Yaskawa INFORM job: DEMO_ROOF_SIDE_0625_3PAINT_27.JBI

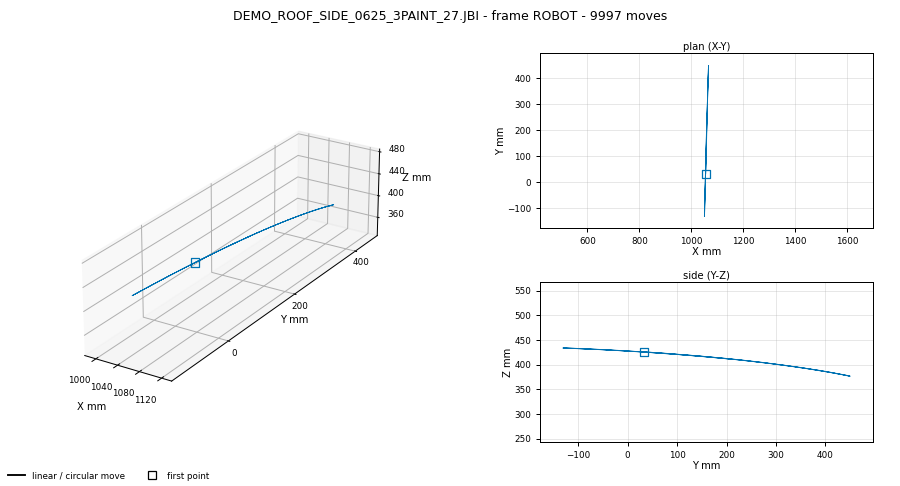
[picture p0: tool path of DEMO_ROOF_SIDE_0625_3PAINT_27.JBI in frame ROBOT, 9997 of 9997 moves have a stored position in this frame; points joined in program order, loops and branches not executed]
/JOB
//NAME DEMO_ROOF_SIDE_0625_3PAINT27
//POS
///NPOS 9997,0,0,0,0,0
///TOOL 0
///USER 0
///POSTYPE ROBOT
///RECTAN
///RCONF 1,0,0,0,0,0,0,0,0,0,0,0,0,0,0,0,0,0,0,0,0,0,0,0
C00000=1055.838,33.048,426.241,171.218,30.645,155.735
C00001=1055.844,33.297,426.225,171.220,30.647,155.735
C00002=1055.850,33.546,426.209,171.221,30.649,155.735
C00003=1055.856,33.796,426.193,171.222,30.652,155.736
C00004=1055.862,34.045,426.176,171.224,30.654,155.736
C00005=1055.869,34.295,426.160,171.225,30.656,155.736
C00006=1055.875,34.544,426.144,171.227,30.658,155.737
C00007=1055.881,34.793,426.128,171.229,30.661,155.737
C00008=1055.887,35.043,426.111,171.230,30.663,155.737
C00009=1055.893,35.292,426.095,171.231,30.665,155.738
C00010=1055.900,35.541,426.080,171.233,30.667,155.738
C00011=1055.906,35.790,426.063,171.235,30.670,155.738
C00012=1055.912,36.040,426.047,171.237,30.672,155.739
C00013=1055.918,36.290,426.030,171.237,30.674,155.739
C00014=1055.924,36.539,426.014,171.239,30.676,155.739
C00015=1055.930,36.789,425.998,171.241,30.679,155.740
C00016=1055.937,37.038,425.982,171.243,30.681,155.740
C00017=1055.943,37.287,425.966,171.244,30.683,155.740
C00018=1055.950,37.537,425.949,171.246,30.686,155.741
C00019=1055.955,37.786,425.933,171.247,30.688,155.741
C00020=1055.961,38.036,425.917,171.248,30.690,155.741
C00021=1055.967,38.285,425.901,171.250,30.693,155.742
C00022=1055.973,38.534,425.884,171.252,30.695,155.742
C00023=1055.979,38.784,425.868,171.254,30.698,155.742
C00024=1055.986,39.033,425.851,171.254,30.699,155.743
C00025=1055.992,39.282,425.835,171.256,30.702,155.743
C00026=1055.998,39.532,425.818,171.258,30.704,155.743
C00027=1056.004,39.781,425.802,171.260,30.706,155.744
C00028=1056.010,40.031,425.786,171.261,30.709,155.744
C00029=1056.016,40.280,425.769,171.263,30.711,155.744
C00030=1056.023,40.529,425.752,171.264,30.714,155.745
C00031=1056.029,40.779,425.736,171.265,30.716,155.745
C00032=1056.035,41.028,425.720,171.267,30.719,155.746
C00033=1056.041,41.277,425.703,171.269,30.721,155.746
C00034=1056.047,41.527,425.687,171.271,30.723,155.746
C00035=1056.053,41.776,425.670,171.271,30.725,155.747
C00036=1056.059,42.025,425.654,171.273,30.727,155.747
C00037=1056.065,42.275,425.637,171.275,30.730,155.747
C00038=1056.071,42.525,425.620,171.276,30.732,155.748
C00039=1056.076,42.774,425.604,171.278,30.735,155.748
C00040=1056.083,43.023,425.587,171.280,30.737,155.748
C00041=1056.089,43.273,425.571,171.281,30.739,155.749
C00042=1056.095,43.522,425.554,171.282,30.742,155.749
C00043=1056.101,43.771,425.538,171.284,30.744,155.749
C00044=1056.108,44.021,425.521,171.286,30.746,155.750
C00045=1056.113,44.270,425.504,171.287,30.748,155.750
C00046=1056.119,44.520,425.488,171.288,30.751,155.750
C00047=1056.125,44.768,425.471,171.290,30.754,155.751
C00048=1056.131,45.018,425.454,171.292,30.756,155.751
C00049=1056.137,45.268,425.437,171.293,30.759,155.752
C00050=1056.144,45.553,425.418,171.295,30.761,155.752
C00051=1056.151,45.838,425.399,171.296,30.764,155.752
C00052=1056.158,46.123,425.380,171.298,30.767,155.753
C00053=1056.164,46.410,425.360,171.300,30.769,155.753
C00054=1056.171,46.659,425.343,171.302,30.772,155.753
C00055=1056.177,46.908,425.327,171.303,30.774,155.754
C00056=1056.183,47.157,425.310,171.305,30.776,155.754
C00057=1056.189,47.407,425.293,171.306,30.779,155.755
C00058=1056.195,47.656,425.277,171.308,30.782,155.755
C00059=1056.201,47.905,425.260,171.309,30.784,155.755
C00060=1056.206,48.155,425.243,171.311,30.786,155.756
C00061=1056.213,48.404,425.226,171.313,30.788,155.756
C00062=1056.219,48.653,425.209,171.313,30.791,155.756
C00063=1056.225,48.903,425.192,171.315,30.793,155.757
C00064=1056.231,49.153,425.175,171.317,30.796,155.757
C00065=1056.237,49.401,425.158,171.319,30.798,155.757
C00066=1056.243,49.651,425.142,171.320,30.800,155.758
C00067=1056.249,49.900,425.124,171.322,30.803,155.758
C00068=1056.255,50.150,425.108,171.323,30.805,155.758
C00069=1056.262,50.398,425.091,171.324,30.807,155.759
C00070=1056.267,50.648,425.074,171.326,30.810,155.759
C00071=1056.274,50.898,425.057,171.328,30.812,155.759
C00072=1056.280,51.147,425.040,171.329,30.815,155.760
C00073=1056.285,51.396,425.023,171.330,30.817,155.760
C00074=1056.292,51.646,425.006,171.332,30.819,155.761
C00075=1056.298,51.895,424.989,171.334,30.822,155.761
C00076=1056.303,52.144,424.972,171.335,30.824,155.761
C00077=1056.310,52.394,424.955,171.337,30.827,155.762
C00078=1056.316,52.643,424.939,171.339,30.829,155.762
C00079=1056.321,52.892,424.921,171.339,30.831,155.762
C00080=1056.328,53.142,424.904,171.341,30.834,155.763
C00081=1056.334,53.391,424.887,171.343,30.836,155.763
C00082=1056.340,53.640,424.870,171.345,30.838,155.763
C00083=1056.346,53.890,424.853,171.346,30.841,155.764
C00084=1056.352,54.139,424.836,171.347,30.843,155.764
C00085=1056.359,54.389,424.818,171.349,30.846,155.765
C00086=1056.365,54.638,424.802,171.350,30.848,155.765
C00087=1056.370,54.887,424.785,171.352,30.850,155.765
C00088=1056.377,55.136,424.767,171.354,30.853,155.766
C00089=1056.383,55.386,424.751,171.356,30.855,155.766
C00090=1056.389,55.635,424.733,171.356,30.857,155.766
C00091=1056.395,55.884,424.716,171.358,30.860,155.767
C00092=1056.401,56.134,424.700,171.360,30.862,155.767
C00093=1056.407,56.383,424.682,171.361,30.865,155.767
C00094=1056.414,56.632,424.665,171.363,30.867,155.768
C00095=1056.420,56.882,424.648,171.365,30.869,155.768
C00096=1056.426,57.131,424.631,171.366,30.871,155.768
C00097=1056.433,57.381,424.613,171.367,30.873,155.769
C00098=1056.438,57.630,424.597,171.369,30.876,155.769
C00099=1056.444,57.879,424.580,171.371,30.878,155.769
C00100=1056.450,58.129,424.562,171.372,30.881,155.770
C00101=1056.457,58.377,424.545,171.374,30.883,155.770
C00102=1056.463,58.627,424.528,171.375,30.886,155.770
C00103=1056.469,58.876,424.510,171.376,30.888,155.771
C00104=1056.475,59.126,424.493,171.378,30.890,155.771
C00105=1056.481,59.375,424.476,171.380,30.892,155.771
C00106=1056.488,59.624,424.458,171.382,30.895,155.772
C00107=1056.494,59.874,424.442,171.383,30.897,155.772
C00108=1056.500,60.123,424.424,171.384,30.900,155.773
C00109=1056.506,60.372,424.407,171.386,30.902,155.773
C00110=1056.512,60.622,424.389,171.387,30.904,155.773
C00111=1056.519,60.871,424.372,171.389,30.906,155.774
C00112=1056.525,61.121,424.356,171.391,30.909,155.774
C00113=1056.531,61.370,424.338,171.392,30.911,155.774
C00114=1056.539,61.655,424.318,171.394,30.914,155.775
C00115=1056.545,61.940,424.298,171.396,30.917,155.775
C00116=1056.553,62.225,424.278,171.398,30.919,155.775
C00117=1056.559,62.510,424.259,171.399,30.922,155.776
C00118=1056.566,62.760,424.241,171.401,30.924,155.776
C00119=1056.572,63.009,424.224,171.402,30.927,155.777
C00120=1056.579,63.258,424.206,171.404,30.929,155.777
C00121=1056.584,63.507,424.189,171.405,30.931,155.777
C00122=1056.591,63.757,424.171,171.407,30.934,155.778
C00123=1056.596,64.006,424.155,171.409,30.936,155.778
C00124=1056.603,64.256,424.137,171.410,30.938,155.778
C00125=1056.609,64.505,424.120,171.411,30.941,155.779
C00126=1056.615,64.754,424.102,171.413,30.943,155.779
C00127=1056.621,65.003,424.085,171.415,30.946,155.779
C00128=1056.627,65.253,424.067,171.416,30.948,155.780
C00129=1056.634,65.502,424.050,171.418,30.950,155.780
C00130=1056.639,65.751,424.032,171.420,30.953,155.781
C00131=1056.646,66.001,424.014,171.420,30.955,155.781
C00132=1056.652,66.250,423.997,171.422,30.958,155.781
C00133=1056.658,66.500,423.979,171.424,30.960,155.782
C00134=1056.663,66.749,423.962,171.426,30.962,155.782
C00135=1056.670,66.998,423.944,171.427,30.964,155.782
C00136=1056.676,67.247,423.927,171.429,30.967,155.783
C00137=1056.682,67.497,423.909,171.430,30.970,155.783
C00138=1056.688,67.745,423.890,171.431,30.972,155.783
C00139=1056.695,67.995,423.873,171.433,30.974,155.784
C00140=1056.701,68.244,423.855,171.435,30.977,155.784
C00141=1056.706,68.493,423.838,171.436,30.979,155.785
C00142=1056.712,68.743,423.820,171.438,30.981,155.785
C00143=1056.719,68.992,423.803,171.439,30.984,155.785
C00144=1056.725,69.242,423.785,171.441,30.987,155.786
C00145=1056.730,69.491,423.767,171.442,30.989,155.786
C00146=1056.736,69.740,423.749,171.444,30.991,155.786
C00147=1056.743,69.990,423.732,171.446,30.993,155.787
C00148=1056.749,70.238,423.714,171.447,30.996,155.787
C00149=1056.755,70.488,423.696,171.448,30.999,155.788
C00150=1056.761,70.737,423.678,171.450,31.001,155.788
C00151=1056.767,70.987,423.660,171.452,31.003,155.788
C00152=1056.772,71.236,423.643,171.453,31.006,155.789
C00153=1056.779,71.485,423.624,171.455,31.008,155.789
C00154=1056.786,71.734,423.607,171.456,31.011,155.789
C00155=1056.791,71.983,423.589,171.457,31.013,155.790
C00156=1056.797,72.233,423.571,171.459,31.015,155.790
C00157=1056.803,72.482,423.554,171.461,31.018,155.790
C00158=1056.809,72.731,423.535,171.462,31.020,155.791
C00159=1056.815,72.981,423.517,171.464,31.023,155.791
C00160=1056.821,73.230,423.499,171.465,31.025,155.792
C00161=1056.827,73.480,423.482,171.467,31.027,155.792
C00162=1056.834,73.729,423.463,171.468,31.030,155.792
C00163=1056.840,73.978,423.446,171.470,31.032,155.793
C00164=1056.846,74.227,423.428,171.472,31.035,155.793
C00165=1056.851,74.476,423.410,171.473,31.037,155.793
C00166=1056.858,74.726,423.392,171.475,31.039,155.794
C00167=1056.864,74.975,423.374,171.476,31.042,155.794
C00168=1056.869,75.224,423.356,171.477,31.045,155.795
C00169=1056.876,75.474,423.338,171.479,31.047,155.795
C00170=1056.882,75.723,423.320,171.481,31.049,155.795
C00171=1056.887,75.972,423.302,171.483,31.051,155.796
C00172=1056.894,76.221,423.283,171.484,31.054,155.796
C00173=1056.900,76.471,423.266,171.485,31.057,155.796
C00174=1056.906,76.720,423.249,171.487,31.059,155.797
C00175=1056.913,76.969,423.230,171.488,31.061,155.797
C00176=1056.919,77.219,423.212,171.490,31.063,155.797
C00177=1056.925,77.468,423.193,171.492,31.066,155.798
C00178=1056.932,77.752,423.173,171.494,31.069,155.798
C00179=1056.938,78.038,423.152,171.495,31.071,155.799
C00180=1056.945,78.323,423.131,171.497,31.075,155.799
C00181=1056.952,78.608,423.111,171.499,31.077,155.800
C00182=1056.958,78.856,423.093,171.500,31.079,155.800
C00183=1056.964,79.106,423.075,171.502,31.082,155.800
C00184=1056.970,79.356,423.057,171.504,31.085,155.801
C00185=1056.976,79.605,423.037,171.505,31.087,155.801
C00186=1056.982,79.854,423.020,171.506,31.089,155.801
C00187=1056.988,80.103,423.001,171.508,31.092,155.802
C00188=1056.994,80.353,422.983,171.510,31.095,155.802
C00189=1057.000,80.602,422.965,171.511,31.097,155.803
C00190=1057.006,80.851,422.947,171.513,31.099,155.803
C00191=1057.012,81.101,422.928,171.514,31.102,155.803
C00192=1057.017,81.350,422.910,171.515,31.105,155.804
C00193=1057.024,81.599,422.892,171.517,31.107,155.804
C00194=1057.030,81.848,422.873,171.519,31.109,155.805
C00195=1057.036,82.097,422.855,171.521,31.112,155.805
C00196=1057.042,82.346,422.837,171.522,31.114,155.805
C00197=1057.047,82.596,422.818,171.523,31.117,155.806
C00198=1057.054,82.845,422.800,171.525,31.119,155.806
C00199=1057.059,83.094,422.782,171.526,31.121,155.806
C00200=1057.066,83.344,422.763,171.528,31.124,155.807
C00201=1057.072,83.593,422.745,171.530,31.127,155.807
C00202=1057.078,83.842,422.727,171.532,31.129,155.807
C00203=1057.084,84.091,422.708,171.532,31.131,155.808
C00204=1057.090,84.341,422.690,171.534,31.134,155.808
C00205=1057.096,84.590,422.671,171.536,31.136,155.809
C00206=1057.102,84.839,422.653,171.537,31.139,155.809
C00207=1057.108,85.088,422.635,171.539,31.141,155.809
C00208=1057.114,85.338,422.616,171.541,31.143,155.810
C00209=1057.120,85.587,422.597,171.543,31.146,155.810
C00210=1057.126,85.837,422.579,171.543,31.149,155.811
C00211=1057.133,86.086,422.561,171.545,31.151,155.811
C00212=1057.138,86.334,422.542,171.547,31.153,155.811
C00213=1057.144,86.584,422.524,171.548,31.156,155.812
C00214=1057.150,86.833,422.505,171.550,31.158,155.812
C00215=1057.157,87.082,422.486,171.552,31.161,155.812
C00216=1057.163,87.331,422.468,171.553,31.163,155.813
C00217=1057.169,87.582,422.449,171.554,31.165,155.813
C00218=1057.174,87.830,422.431,171.556,31.168,155.814
C00219=1057.181,88.079,422.412,171.558,31.171,155.814
C00220=1057.187,88.329,422.394,171.559,31.173,155.814
C00221=1057.193,88.578,422.376,171.561,31.175,155.815
C00222=1057.199,88.827,422.357,171.562,31.178,155.815
C00223=1057.205,89.076,422.338,171.564,31.180,155.815
C00224=1057.211,89.325,422.320,171.565,31.183,155.816
C00225=1057.217,89.575,422.302,171.567,31.185,155.816
C00226=1057.223,89.824,422.282,171.569,31.187,155.817
C00227=1057.229,90.073,422.264,171.571,31.190,155.817
C00228=1057.236,90.322,422.245,171.572,31.192,155.817
C00229=1057.242,90.571,422.227,171.573,31.195,155.818
C00230=1057.248,90.821,422.208,171.575,31.197,155.818
C00231=1057.254,91.071,422.189,171.576,31.200,155.819
C00232=1057.259,91.319,422.170,171.578,31.202,155.819
C00233=1057.266,91.568,422.152,171.580,31.205,155.819
C00234=1057.271,91.818,422.133,171.582,31.207,155.820
C00235=1057.278,92.067,422.114,171.582,31.210,155.820
C00236=1057.283,92.316,422.095,171.584,31.212,155.820
C00237=1057.290,92.566,422.076,171.586,31.214,155.821
C00238=1057.295,92.814,422.057,171.588,31.217,155.821
C00239=1057.301,93.064,422.039,171.589,31.220,155.822
C00240=1057.307,93.313,422.020,171.591,31.222,155.822
C00241=1057.313,93.563,422.001,171.593,31.224,155.822
C00242=1057.320,93.848,421.979,171.594,31.227,155.823
C00243=1057.327,94.133,421.957,171.596,31.230,155.823
C00244=1057.334,94.417,421.936,171.598,31.233,155.824
C00245=1057.340,94.702,421.915,171.600,31.236,155.824
C00246=1057.346,94.952,421.896,171.601,31.238,155.825
C00247=1057.353,95.201,421.877,171.603,31.241,155.825
C00248=1057.358,95.450,421.858,171.604,31.244,155.825
C00249=1057.365,95.699,421.839,171.606,31.246,155.826
C00250=1057.370,95.949,421.820,171.607,31.248,155.826
C00251=1057.377,96.198,421.801,171.609,31.251,155.826
C00252=1057.382,96.447,421.782,171.611,31.253,155.827
C00253=1057.389,96.696,421.764,171.612,31.255,155.827
C00254=1057.394,96.944,421.744,171.614,31.258,155.828
C00255=1057.401,97.194,421.725,171.615,31.261,155.828
C00256=1057.406,97.443,421.706,171.617,31.263,155.828
C00257=1057.413,97.692,421.687,171.618,31.265,155.829
C00258=1057.418,97.942,421.668,171.620,31.268,155.829
C00259=1057.425,98.191,421.649,171.622,31.270,155.829
C00260=1057.431,98.440,421.630,171.624,31.273,155.830
C00261=1057.437,98.689,421.612,171.624,31.275,155.830
C00262=1057.443,98.939,421.592,171.626,31.278,155.831
C00263=1057.449,99.188,421.574,171.628,31.280,155.831
C00264=1057.455,99.437,421.554,171.630,31.283,155.831
C00265=1057.461,99.686,421.535,171.631,31.285,155.832
C00266=1057.467,99.935,421.516,171.633,31.287,155.832
C00267=1057.473,100.185,421.497,171.635,31.290,155.833
C00268=1057.479,100.434,421.478,171.636,31.293,155.833
C00269=1057.485,100.683,421.459,171.637,31.295,155.833
C00270=1057.491,100.932,421.440,171.639,31.297,155.834
C00271=1057.497,101.181,421.420,171.641,31.300,155.834
C00272=1057.503,101.431,421.401,171.643,31.303,155.835
C00273=1057.509,101.680,421.382,171.644,31.305,155.835
C00274=1057.515,101.929,421.363,171.646,31.307,155.835
C00275=1057.521,102.178,421.343,171.647,31.310,155.836
C00276=1057.527,102.427,421.324,171.649,31.313,155.836
C00277=1057.533,102.677,421.305,171.650,31.315,155.837
C00278=1057.539,102.926,421.286,171.652,31.318,155.837
C00279=1057.545,103.175,421.266,171.654,31.320,155.837
C00280=1057.551,103.424,421.247,171.656,31.322,155.838
C00281=1057.556,103.674,421.227,171.657,31.325,155.838
C00282=1057.562,103.923,421.208,171.658,31.328,155.839
C00283=1057.569,104.172,421.189,171.660,31.330,155.839
C00284=1057.575,104.421,421.170,171.662,31.332,155.839
C00285=1057.580,104.670,421.150,171.663,31.335,155.840
C00286=1057.586,104.919,421.130,171.665,31.338,155.840
C00287=1057.592,105.169,421.111,171.667,31.340,155.840
C00288=1057.598,105.418,421.092,171.669,31.343,155.841
C00289=1057.604,105.667,421.073,171.669,31.345,155.841
C00290=1057.610,105.916,421.053,171.671,31.348,155.842
C00291=1057.616,106.165,421.033,171.673,31.350,155.842
C00292=1057.622,106.414,421.014,171.675,31.353,155.842
C00293=1057.628,106.663,420.995,171.676,31.355,155.843
C00294=1057.634,106.912,420.975,171.678,31.357,155.843
C00295=1057.640,107.162,420.956,171.680,31.360,155.844
C00296=1057.646,107.410,420.936,171.681,31.363,155.844
C00297=1057.651,107.660,420.917,171.682,31.365,155.844
C00298=1057.659,107.910,420.898,171.684,31.367,155.845
C00299=1057.665,108.158,420.878,171.686,31.370,155.845
C00300=1057.670,108.408,420.859,171.688,31.373,155.846
C00301=1057.676,108.657,420.839,171.689,31.375,155.846
C00302=1057.682,108.906,420.820,171.691,31.377,155.846
C00303=1057.688,109.155,420.800,171.692,31.380,155.847
C00304=1057.694,109.404,420.781,171.694,31.383,155.847
C00305=1057.700,109.653,420.761,171.695,31.385,155.848
C00306=1057.707,109.938,420.739,171.698,31.388,155.848
C00307=1057.714,110.224,420.716,171.700,31.391,155.848
C00308=1057.721,110.508,420.693,171.702,31.393,155.849
C00309=1057.728,110.793,420.671,171.703,31.396,155.849
C00310=1057.734,111.042,420.652,171.704,31.398,155.850
C00311=1057.740,111.292,420.632,171.706,31.401,155.850
C00312=1057.745,111.540,420.612,171.708,31.404,155.850
C00313=1057.751,111.790,420.593,171.710,31.406,155.851
C00314=1057.757,112.039,420.573,171.711,31.409,155.851
C00315=1057.763,112.289,420.553,171.713,31.411,155.852
C00316=1057.769,112.538,420.534,171.714,31.414,155.852
C00317=1057.775,112.786,420.514,171.716,31.416,155.852
C00318=1057.781,113.036,420.494,171.718,31.419,155.853
C00319=1057.787,113.285,420.474,171.719,31.421,155.853
C00320=1057.793,113.534,420.455,171.721,31.423,155.854
C00321=1057.799,113.783,420.435,171.723,31.426,155.854
C00322=1057.805,114.032,420.415,171.725,31.429,155.854
C00323=1057.811,114.282,420.396,171.726,31.431,155.855
C00324=1057.817,114.531,420.376,171.727,31.434,155.855
C00325=1057.823,114.779,420.356,171.729,31.437,155.856
C00326=1057.829,115.029,420.336,171.731,31.439,155.856
C00327=1057.834,115.278,420.316,171.733,31.442,155.857
C00328=1057.840,115.527,420.296,171.734,31.444,155.857
C00329=1057.846,115.776,420.276,171.736,31.446,155.857
C00330=1057.852,116.026,420.256,171.738,31.449,155.858
C00331=1057.858,116.275,420.236,171.739,31.452,155.858
C00332=1057.864,116.524,420.216,171.740,31.454,155.859
C00333=1057.870,116.772,420.196,171.742,31.457,155.859
C00334=1057.875,117.022,420.177,171.744,31.460,155.859
C00335=1057.881,117.271,420.157,171.746,31.462,155.860
C00336=1057.887,117.521,420.136,171.748,31.465,155.860
C00337=1057.893,117.769,420.116,171.749,31.467,155.861
C00338=1057.899,118.018,420.096,171.750,31.470,155.861
C00339=1057.905,118.268,420.077,171.752,31.472,155.861
C00340=1057.910,118.517,420.056,171.754,31.475,155.862
C00341=1057.916,118.766,420.036,171.756,31.477,155.862
C00342=1057.923,119.015,420.016,171.757,31.480,155.863
C00343=1057.929,119.264,419.996,171.759,31.483,155.863
C00344=1057.934,119.513,419.975,171.761,31.485,155.863
C00345=1057.940,119.762,419.956,171.762,31.488,155.864
C00346=1057.946,120.011,419.936,171.764,31.491,155.864
C00347=1057.952,120.261,419.916,171.765,31.493,155.865
C00348=1057.957,120.510,419.895,171.767,31.495,155.865
C00349=1057.963,120.759,419.875,171.769,31.498,155.865
C00350=1057.969,121.008,419.855,171.771,31.500,155.866
C00351=1057.976,121.257,419.835,171.773,31.503,155.866
C00352=1057.981,121.506,419.814,171.774,31.506,155.867
C00353=1057.987,121.755,419.794,171.775,31.508,155.867
C00354=1057.993,122.004,419.774,171.777,31.511,155.868
C00355=1057.999,122.254,419.754,171.779,31.513,155.868
C00356=1058.005,122.502,419.734,171.781,31.516,155.868
C00357=1058.011,122.751,419.714,171.782,31.518,155.869
C00358=1058.017,123.000,419.694,171.784,31.521,155.869
C00359=1058.023,123.250,419.673,171.786,31.523,155.870
C00360=1058.029,123.499,419.654,171.787,31.526,155.870
C00361=1058.035,123.748,419.634,171.789,31.529,155.870
C00362=1058.040,123.998,419.613,171.790,31.531,155.871
C00363=1058.047,124.246,419.592,171.792,31.533,155.871
C00364=1058.053,124.495,419.572,171.794,31.536,155.872
C00365=1058.059,124.744,419.552,171.796,31.539,155.872
C00366=1058.065,124.994,419.531,171.798,31.541,155.872
C00367=1058.071,125.242,419.511,171.800,31.544,155.873
C00368=1058.077,125.491,419.491,171.800,31.546,155.873
C00369=1058.082,125.741,419.470,171.802,31.548,155.874
C00370=1058.090,126.025,419.448,171.804,31.552,155.874
C00371=1058.096,126.310,419.424,171.806,31.554,155.874
C00372=1058.103,126.595,419.401,171.809,31.558,155.875
C00373=1058.110,126.880,419.378,171.811,31.560,155.875
C00374=1058.116,127.130,419.357,171.812,31.563,155.876
C00375=1058.122,127.378,419.337,171.813,31.565,155.876
C00376=1058.128,127.627,419.317,171.815,31.567,155.877
C00377=1058.134,127.877,419.296,171.817,31.570,155.877
C00378=1058.140,128.126,419.276,171.819,31.573,155.877
C00379=1058.146,128.374,419.256,171.821,31.575,155.878
C00380=1058.152,128.624,419.235,171.823,31.578,155.878
C00381=1058.158,128.873,419.215,171.824,31.580,155.879
C00382=1058.165,129.122,419.194,171.826,31.583,155.879
C00383=1058.170,129.371,419.174,171.827,31.585,155.879
C00384=1058.176,129.620,419.153,171.829,31.588,155.880
C00385=1058.182,129.869,419.132,171.831,31.591,155.880
C00386=1058.188,130.118,419.112,171.833,31.593,155.881
C00387=1058.195,130.368,419.092,171.834,31.595,155.881
C00388=1058.200,130.617,419.071,171.836,31.598,155.881
C00389=1058.207,130.866,419.050,171.838,31.600,155.882
C00390=1058.213,131.115,419.030,171.840,31.603,155.882
C00391=1058.218,131.364,419.010,171.841,31.606,155.883
C00392=1058.225,131.613,418.989,171.843,31.608,155.883
C00393=1058.230,131.862,418.968,171.845,31.610,155.883
C00394=1058.237,132.111,418.948,171.846,31.613,155.884
C00395=1058.242,132.360,418.927,171.848,31.615,155.884
C00396=1058.248,132.609,418.907,171.850,31.618,155.885
C00397=1058.254,132.858,418.886,171.852,31.621,155.885
C00398=1058.259,133.107,418.865,171.854,31.623,155.885
C00399=1058.266,133.356,418.844,171.855,31.626,155.886
C00400=1058.272,133.606,418.824,171.857,31.629,155.886
C00401=1058.277,133.855,418.803,171.858,31.631,155.887
C00402=1058.284,134.104,418.782,171.860,31.634,155.887
C00403=1058.289,134.353,418.761,171.862,31.636,155.888
C00404=1058.296,134.602,418.740,171.864,31.639,155.888
C00405=1058.301,134.851,418.720,171.866,31.642,155.888
C00406=1058.307,135.100,418.698,171.868,31.644,155.889
C00407=1058.313,135.349,418.678,171.869,31.646,155.889
C00408=1058.319,135.599,418.657,171.871,31.649,155.890
C00409=1058.325,135.847,418.636,171.872,31.652,155.890
C00410=1058.331,136.096,418.616,171.874,31.654,155.890
C00411=1058.337,136.345,418.594,171.876,31.657,155.891
C00412=1058.342,136.594,418.574,171.878,31.659,155.891
C00413=1058.349,136.843,418.553,171.880,31.662,155.892
C00414=1058.354,137.092,418.532,171.882,31.665,155.892
C00415=1058.360,137.341,418.511,171.883,31.667,155.893
C00416=1058.366,137.590,418.491,171.885,31.670,155.893
C00417=1058.373,137.839,418.469,171.886,31.672,155.893
C00418=1058.378,138.089,418.449,171.888,31.675,155.894
C00419=1058.385,138.337,418.428,171.890,31.678,155.894
C00420=1058.390,138.587,418.407,171.892,31.680,155.895
C00421=1058.396,138.836,418.385,171.894,31.682,155.895
C00422=1058.401,139.085,418.365,171.896,31.685,155.895
C00423=1058.408,139.334,418.344,171.897,31.688,155.896
C00424=1058.414,139.582,418.322,171.899,31.690,155.896
C00425=1058.420,139.832,418.302,171.901,31.693,155.897
C00426=1058.425,140.081,418.280,171.902,31.695,155.897
C00427=1058.432,140.330,418.260,171.904,31.698,155.897
C00428=1058.437,140.579,418.239,171.906,31.701,155.898
C00429=1058.444,140.828,418.217,171.908,31.703,155.898
C00430=1058.449,141.077,418.196,171.910,31.706,155.899
C00431=1058.455,141.326,418.175,171.911,31.709,155.899
C00432=1058.461,141.575,418.154,171.913,31.711,155.900
C00433=1058.466,141.824,418.133,171.915,31.714,155.900
C00434=1058.474,142.109,418.108,171.917,31.717,155.901
C00435=1058.481,142.393,418.084,171.919,31.720,155.901
C00436=1058.487,142.678,418.059,171.921,31.723,155.901
C00437=1058.493,142.963,418.036,171.923,31.726,155.902
C00438=1058.500,143.212,418.014,171.925,31.728,155.902
C00439=1058.505,143.461,417.993,171.926,31.731,155.903
C00440=1058.511,143.710,417.971,171.928,31.733,155.903
C00441=1058.517,143.959,417.951,171.930,31.736,155.904
C00442=1058.523,144.208,417.929,171.932,31.739,155.904
C00443=1058.530,144.457,417.908,171.934,31.741,155.904
C00444=1058.535,144.706,417.887,171.936,31.744,155.905
C00445=1058.541,144.956,417.866,171.938,31.747,155.905
C00446=1058.547,145.204,417.845,171.940,31.749,155.906
C00447=1058.553,145.453,417.823,171.942,31.752,155.906
C00448=1058.559,145.702,417.802,171.942,31.754,155.907
C00449=1058.565,145.951,417.780,171.944,31.757,155.907
C00450=1058.571,146.200,417.759,171.946,31.760,155.907
C00451=1058.576,146.449,417.738,171.948,31.762,155.908
C00452=1058.582,146.698,417.716,171.950,31.765,155.908
C00453=1058.588,146.948,417.695,171.952,31.767,155.909
C00454=1058.594,147.196,417.674,171.954,31.770,155.909
C00455=1058.600,147.445,417.652,171.956,31.773,155.910
C00456=1058.607,147.694,417.631,171.957,31.775,155.910
C00457=1058.612,147.943,417.609,171.959,31.778,155.910
C00458=1058.618,148.192,417.587,171.961,31.781,155.911
C00459=1058.623,148.441,417.567,171.963,31.783,155.911
C00460=1058.629,148.691,417.545,171.965,31.786,155.912
C00461=1058.636,148.940,417.524,171.967,31.788,155.912
C00462=1058.641,149.188,417.502,171.969,31.791,155.912
C00463=1058.647,149.438,417.481,171.971,31.794,155.913
C00464=1058.653,149.687,417.459,171.972,31.797,155.913
C00465=1058.659,149.935,417.438,171.973,31.799,155.914
C00466=1058.665,150.184,417.416,171.975,31.802,155.914
C00467=1058.671,150.434,417.394,171.977,31.805,155.915
C00468=1058.676,150.683,417.373,171.979,31.807,155.915
C00469=1058.682,150.932,417.351,171.981,31.810,155.916
C00470=1058.688,151.181,417.329,171.983,31.813,155.916
C00471=1058.694,151.429,417.308,171.985,31.815,155.916
C00472=1058.700,151.679,417.286,171.987,31.818,155.917
C00473=1058.707,151.927,417.264,171.989,31.820,155.917
C00474=1058.711,152.176,417.242,171.990,31.823,155.918
C00475=1058.718,152.425,417.221,171.992,31.826,155.918
C00476=1058.724,152.674,417.199,171.994,31.828,155.919
C00477=1058.729,152.923,417.178,171.996,31.831,155.919
C00478=1058.736,153.172,417.156,171.998,31.834,155.919
C00479=1058.742,153.421,417.134,172.000,31.837,155.920
C00480=1058.747,153.671,417.112,172.002,31.839,155.920
C00481=1058.753,153.919,417.091,172.004,31.842,155.921
C00482=1058.759,154.168,417.069,172.005,31.845,155.921
C00483=1058.765,154.417,417.047,172.007,31.847,155.922
C00484=1058.771,154.666,417.026,172.009,31.850,155.922
C00485=1058.776,154.915,417.003,172.011,31.852,155.922
C00486=1058.782,155.164,416.982,172.013,31.855,155.923
C00487=1058.789,155.414,416.960,172.015,31.858,155.923
C00488=1058.794,155.661,416.938,172.017,31.860,155.924
C00489=1058.800,155.911,416.916,172.019,31.863,155.924
C00490=1058.806,156.160,416.894,172.021,31.866,155.925
C00491=1058.812,156.409,416.873,172.022,31.869,155.925
C00492=1058.817,156.658,416.850,172.024,31.871,155.926
C00493=1058.824,156.907,416.828,172.026,31.874,155.926
C00494=1058.830,157.156,416.807,172.028,31.877,155.926
C00495=1058.835,157.406,416.785,172.029,31.879,155.927
C00496=1058.841,157.653,416.763,172.031,31.882,155.927
C00497=1058.847,157.903,416.741,172.033,31.884,155.928
C00498=1058.854,158.187,416.715,172.036,31.888,155.928
C00499=1058.861,158.472,416.690,172.038,31.891,155.929
C00500=1058.867,158.756,416.665,172.039,31.894,155.929
C00501=1058.874,159.041,416.641,172.042,31.897,155.930
C00502=1058.880,159.290,416.618,172.044,31.899,155.930
C00503=1058.885,159.538,416.596,172.046,31.902,155.931
C00504=1058.892,159.787,416.574,172.048,31.905,155.931
C00505=1058.897,160.036,416.552,172.050,31.908,155.931
C00506=1058.904,160.285,416.530,172.052,31.910,155.932
C00507=1058.910,160.534,416.508,172.054,31.913,155.932
C00508=1058.915,160.783,416.486,172.056,31.916,155.933
C00509=1058.921,161.031,416.464,172.058,31.918,155.933
C00510=1058.927,161.281,416.441,172.059,31.921,155.934
C00511=1058.932,161.530,416.418,172.061,31.924,155.934
C00512=1058.939,161.779,416.397,172.063,31.927,155.935
C00513=1058.944,162.027,416.374,172.065,31.929,155.935
C00514=1058.949,162.277,416.352,172.067,31.932,155.936
C00515=1058.956,162.525,416.330,172.069,31.935,155.936
C00516=1058.961,162.775,416.307,172.071,31.938,155.936
C00517=1058.967,163.024,416.284,172.073,31.941,155.937
C00518=1058.972,163.272,416.263,172.075,31.943,155.937
C00519=1058.978,163.521,416.240,172.076,31.946,155.938
C00520=1058.984,163.771,416.218,172.078,31.949,155.938
C00521=1058.989,164.019,416.195,172.080,31.952,155.939
C00522=1058.995,164.269,416.173,172.082,31.954,155.939
C00523=1059.001,164.517,416.151,172.084,31.958,155.940
C00524=1059.006,164.766,416.128,172.086,31.960,155.940
C00525=1059.012,165.015,416.106,172.088,31.963,155.941
C00526=1059.018,165.264,416.083,172.090,31.966,155.941
C00527=1059.024,165.513,416.060,172.092,31.969,155.942
C00528=1059.029,165.762,416.039,172.093,31.971,155.942
C00529=1059.035,166.010,416.016,172.095,31.974,155.942
C00530=1059.041,166.259,415.993,172.097,31.977,155.943
C00531=1059.046,166.509,415.971,172.099,31.980,155.943
C00532=1059.052,166.758,415.948,172.101,31.982,155.944
C00533=1059.059,167.006,415.926,172.103,31.985,155.944
C00534=1059.064,167.256,415.903,172.105,31.988,155.945
C00535=1059.070,167.505,415.881,172.107,31.991,155.945
C00536=1059.075,167.753,415.858,172.109,31.994,155.946
C00537=1059.081,168.002,415.836,172.111,31.996,155.946
C00538=1059.087,168.251,415.813,172.113,31.999,155.947
C00539=1059.092,168.500,415.790,172.115,32.002,155.947
C00540=1059.098,168.749,415.767,172.117,32.005,155.948
C00541=1059.105,168.997,415.745,172.119,32.008,155.948
C00542=1059.110,169.247,415.723,172.121,32.010,155.948
C00543=1059.116,169.496,415.700,172.123,32.013,155.949
C00544=1059.122,169.744,415.677,172.125,32.016,155.949
C00545=1059.128,169.993,415.655,172.127,32.019,155.950
C00546=1059.134,170.242,415.632,172.129,32.022,155.950
C00547=1059.139,170.491,415.609,172.131,32.024,155.951
C00548=1059.145,170.740,415.587,172.132,32.027,155.951
C00549=1059.151,170.989,415.564,172.134,32.030,155.952
C00550=1059.156,171.237,415.542,172.136,32.033,155.952
C00551=1059.162,171.486,415.519,172.139,32.035,155.953
C00552=1059.168,171.735,415.496,172.141,32.038,155.953
C00553=1059.174,171.984,415.473,172.143,32.041,155.954
C00554=1059.179,172.233,415.451,172.145,32.044,155.954
C00555=1059.186,172.482,415.428,172.147,32.046,155.954
C00556=1059.191,172.731,415.405,172.149,32.050,155.955
C00557=1059.197,172.980,415.382,172.151,32.052,155.955
C00558=1059.203,173.229,415.359,172.152,32.055,155.956
C00559=1059.209,173.478,415.336,172.154,32.058,155.956
C00560=1059.215,173.726,415.314,172.156,32.061,155.957
C00561=1059.221,173.976,415.291,172.159,32.063,155.957
C00562=1059.228,174.259,415.265,172.161,32.067,155.958
C00563=1059.234,174.544,415.238,172.163,32.070,155.958
C00564=1059.241,174.828,415.213,172.166,32.073,155.959
C00565=1059.248,175.111,415.187,172.168,32.076,155.959
C00566=1059.254,175.361,415.163,172.170,32.079,155.960
C00567=1059.260,175.610,415.140,172.172,32.081,155.960
C00568=1059.265,175.859,415.118,172.174,32.085,155.961
C00569=1059.272,176.107,415.095,172.176,32.087,155.961
C00570=1059.278,176.356,415.072,172.178,32.090,155.962
C00571=1059.283,176.605,415.049,172.180,32.093,155.962
C00572=1059.289,176.854,415.026,172.182,32.096,155.963
C00573=1059.295,177.103,415.003,172.184,32.098,155.963
C00574=1059.301,177.351,414.980,172.186,32.101,155.963
C00575=1059.306,177.600,414.957,172.189,32.104,155.964
C00576=1059.314,177.849,414.934,172.191,32.107,155.964
C00577=1059.319,178.098,414.911,172.193,32.109,155.965
C00578=1059.325,178.347,414.888,172.195,32.113,155.965
C00579=1059.331,178.596,414.865,172.196,32.115,155.966
C00580=1059.336,178.845,414.842,172.198,32.118,155.966
C00581=1059.343,179.093,414.819,172.200,32.121,155.967
C00582=1059.348,179.342,414.796,172.203,32.124,155.967
C00583=1059.355,179.591,414.773,172.205,32.126,155.968
C00584=1059.361,179.840,414.750,172.207,32.129,155.968
C00585=1059.367,180.089,414.727,172.209,32.132,155.969
C00586=1059.373,180.337,414.703,172.211,32.135,155.969
C00587=1059.379,180.586,414.680,172.213,32.138,155.969
C00588=1059.385,180.836,414.657,172.216,32.140,155.970
C00589=1059.391,181.085,414.634,172.218,32.143,155.970
C00590=1059.396,181.334,414.611,172.219,32.146,155.971
C00591=1059.402,181.582,414.588,172.221,32.149,155.971
C00592=1059.408,181.831,414.565,172.223,32.151,155.972
C00593=1059.415,182.080,414.542,172.226,32.154,155.972
C00594=1059.421,182.328,414.518,172.228,32.157,155.973
C00595=1059.427,182.577,414.495,172.230,32.160,155.973
C00596=1059.433,182.826,414.472,172.232,32.162,155.974
C00597=1059.439,183.075,414.448,172.234,32.166,155.974
C00598=1059.445,183.324,414.425,172.237,32.168,155.975
C00599=1059.451,183.573,414.402,172.239,32.171,155.975
C00600=1059.457,183.821,414.379,172.241,32.174,155.975
C00601=1059.463,184.071,414.355,172.242,32.177,155.976
C00602=1059.469,184.320,414.333,172.244,32.179,155.976
C00603=1059.475,184.568,414.309,172.247,32.183,155.977
C00604=1059.481,184.817,414.286,172.249,32.185,155.977
C00605=1059.487,185.066,414.261,172.251,32.188,155.978
C00606=1059.492,185.315,414.238,172.253,32.191,155.978
C00607=1059.498,185.563,414.215,172.255,32.194,155.979
C00608=1059.503,185.813,414.191,172.257,32.197,155.979
C00609=1059.509,186.061,414.167,172.260,32.200,155.980
C00610=1059.514,186.310,414.144,172.262,32.203,155.980
C00611=1059.521,186.559,414.120,172.264,32.206,155.981
C00612=1059.527,186.808,414.097,172.265,32.209,155.981
C00613=1059.532,187.056,414.073,172.267,32.212,155.982
C00614=1059.538,187.305,414.050,172.270,32.215,155.982
C00615=1059.543,187.554,414.026,172.272,32.218,155.983
C00616=1059.550,187.803,414.001,172.274,32.221,155.983
C00617=1059.555,188.052,413.979,172.276,32.224,155.984
C00618=1059.561,188.300,413.954,172.278,32.227,155.984
C00619=1059.566,188.549,413.931,172.281,32.230,155.985
C00620=1059.572,188.798,413.907,172.283,32.233,155.985
C00621=1059.578,189.047,413.883,172.285,32.236,155.986
C00622=1059.583,189.296,413.860,172.287,32.239,155.986
C00623=1059.589,189.544,413.836,172.290,32.242,155.987
C00624=1059.595,189.793,413.812,172.291,32.245,155.987
C00625=1059.601,190.043,413.788,172.293,32.247,155.988
C00626=1059.608,190.326,413.761,172.296,32.251,155.988
C00627=1059.614,190.609,413.735,172.298,32.254,155.989
C00628=1059.621,190.893,413.707,172.301,32.258,155.990
C00629=1059.628,191.177,413.680,172.303,32.262,155.990
C00630=1059.633,191.425,413.656,172.305,32.264,155.991
C00631=1059.639,191.674,413.632,172.308,32.267,155.991
C00632=1059.646,191.923,413.608,172.310,32.271,155.992
C00633=1059.651,192.171,413.584,172.312,32.273,155.992
C00634=1059.657,192.420,413.561,172.314,32.276,155.993
C00635=1059.662,192.669,413.536,172.317,32.279,155.993
C00636=1059.669,192.918,413.512,172.318,32.282,155.994
C00637=1059.674,193.166,413.488,172.320,32.285,155.994
C00638=1059.680,193.415,413.464,172.322,32.288,155.995
C00639=1059.685,193.664,413.441,172.325,32.291,155.995
C00640=1059.692,193.913,413.417,172.327,32.294,155.996
C00641=1059.697,194.162,413.392,172.329,32.297,155.996
C00642=1059.703,194.410,413.369,172.332,32.300,155.997
C00643=1059.709,194.660,413.344,172.334,32.303,155.997
C00644=1059.715,194.908,413.320,172.336,32.306,155.998
C00645=1059.721,195.156,413.296,172.338,32.309,155.998
C00646=1059.727,195.405,413.272,172.341,32.312,155.999
C00647=1059.732,195.655,413.249,172.343,32.315,155.999
C00648=1059.739,195.904,413.225,172.344,32.318,156.000
C00649=1059.744,196.152,413.200,172.347,32.321,156.000
C00650=1059.751,196.401,413.176,172.349,32.324,156.001
C00651=1059.756,196.650,413.152,172.351,32.327,156.001
C00652=1059.762,196.898,413.128,172.353,32.330,156.002
C00653=1059.768,197.147,413.104,172.356,32.333,156.002
C00654=1059.774,197.396,413.080,172.358,32.336,156.003
C00655=1059.780,197.645,413.055,172.360,32.339,156.003
C00656=1059.786,197.893,413.032,172.363,32.342,156.004
C00657=1059.792,198.143,413.007,172.365,32.345,156.004
C00658=1059.798,198.391,412.983,172.367,32.348,156.005
C00659=1059.804,198.640,412.959,172.370,32.351,156.005
C00660=1059.810,198.888,412.935,172.372,32.354,156.006
C00661=1059.816,199.137,412.910,172.374,32.357,156.006
C00662=1059.822,199.385,412.886,172.376,32.360,156.007
C00663=1059.828,199.635,412.862,172.378,32.363,156.007
C00664=1059.833,199.883,412.837,172.380,32.366,156.008
C00665=1059.840,200.132,412.813,172.383,32.369,156.008
C00666=1059.845,200.381,412.789,172.385,32.372,156.009
C00667=1059.852,200.630,412.765,172.387,32.375,156.009
C00668=1059.857,200.878,412.741,172.390,32.378,156.010
C00669=1059.864,201.127,412.716,172.392,32.381,156.010
C00670=1059.870,201.376,412.691,172.394,32.384,156.011
C00671=1059.876,201.624,412.668,172.397,32.387,156.011
C00672=1059.882,201.874,412.643,172.399,32.391,156.012
C00673=1059.887,202.122,412.619,172.401,32.393,156.012
C00674=1059.894,202.371,412.594,172.404,32.396,156.013
C00675=1059.900,202.619,412.570,172.405,32.400,156.014
C00676=1059.905,202.868,412.545,172.407,32.403,156.014
C00677=1059.911,203.117,412.521,172.410,32.406,156.015
C00678=1059.917,203.366,412.496,172.412,32.409,156.015
C00679=1059.922,203.614,412.471,172.415,32.412,156.016
C00680=1059.928,203.863,412.447,172.417,32.415,156.016
C00681=1059.934,204.111,412.422,172.419,32.419,156.017
C00682=1059.940,204.360,412.398,172.422,32.421,156.017
C00683=1059.946,204.610,412.373,172.424,32.424,156.018
C00684=1059.952,204.858,412.348,172.426,32.428,156.018
C00685=1059.958,205.107,412.324,172.429,32.431,156.019
C00686=1059.963,205.355,412.299,172.431,32.434,156.019
C00687=1059.969,205.604,412.274,172.433,32.437,156.020
C00688=1059.975,205.853,412.250,172.436,32.440,156.021
C00689=1059.982,206.101,412.225,172.438,32.444,156.021
C00690=1060.006,207.150,412.121,172.620,32.529,156.031
C00691=1060.012,207.381,412.097,172.622,32.533,156.031
C00692=1060.017,207.611,412.073,172.623,32.536,156.032
C00693=1060.023,207.842,412.050,172.625,32.540,156.033
C00694=1060.029,208.072,412.026,172.627,32.543,156.033
C00695=1060.035,208.302,412.002,172.629,32.547,156.034
C00696=1060.040,208.532,411.978,172.631,32.551,156.035
C00697=1060.046,208.763,411.954,172.633,32.555,156.036
C00698=1060.052,208.993,411.931,172.633,32.559,156.036
C00699=1060.057,209.242,411.905,172.635,32.562,156.037
C00700=1060.064,209.490,411.879,172.637,32.567,156.038
C00701=1060.070,209.740,411.854,172.639,32.570,156.038
C00702=1060.077,209.988,411.828,172.641,32.575,156.039
C00703=1060.082,210.237,411.802,172.643,32.578,156.040
C00704=1060.089,210.485,411.776,172.645,32.583,156.041
C00705=1060.095,210.734,411.751,172.647,32.586,156.041
C00706=1060.101,210.982,411.725,172.649,32.591,156.042
C00707=1060.107,211.231,411.699,172.651,32.594,156.043
C00708=1060.113,211.480,411.674,172.653,32.599,156.044
C00709=1060.120,211.728,411.648,172.656,32.602,156.044
C00710=1060.125,211.977,411.622,172.658,32.607,156.045
C00711=1060.131,212.225,411.596,172.660,32.610,156.046
C00712=1060.138,212.473,411.570,172.662,32.615,156.047
C00713=1060.143,212.722,411.544,172.664,32.618,156.047
C00714=1060.150,212.971,411.518,172.666,32.623,156.048
C00715=1060.156,213.220,411.492,172.668,32.626,156.049
C00716=1060.162,213.468,411.466,172.670,32.630,156.049
C00717=1060.168,213.717,411.440,172.672,32.634,156.050
C00718=1060.174,213.965,411.414,172.674,32.638,156.051
C00719=1060.180,214.214,411.388,172.676,32.642,156.052
C00720=1060.186,214.462,411.362,172.677,32.646,156.052
C00721=1060.192,214.711,411.336,172.679,32.650,156.053
C00722=1060.198,214.959,411.310,172.681,32.654,156.054
C00723=1060.204,215.208,411.285,172.683,32.658,156.055
C00724=1060.211,215.457,411.258,172.685,32.662,156.055
C00725=1060.217,215.706,411.232,172.687,32.666,156.056
C00726=1060.223,215.954,411.206,172.689,32.670,156.057
C00727=1060.229,216.202,411.180,172.691,32.674,156.058
C00728=1060.235,216.451,411.154,172.693,32.678,156.058
C00729=1060.241,216.699,411.128,172.695,32.682,156.059
C00730=1060.247,216.949,411.101,172.697,32.686,156.060
C00731=1060.254,217.197,411.075,172.699,32.690,156.061
C00732=1060.260,217.445,411.049,172.701,32.694,156.061
C00733=1060.265,217.694,411.023,172.703,32.698,156.062
C00734=1060.272,217.942,410.997,172.706,32.702,156.063
C00735=1060.278,218.191,410.970,172.708,32.706,156.063
C00736=1060.284,218.440,410.944,172.710,32.709,156.064
C00737=1060.290,218.688,410.918,172.712,32.714,156.065
C00738=1060.296,218.936,410.891,172.714,32.717,156.066
C00739=1060.302,219.185,410.866,172.716,32.721,156.066
C00740=1060.309,219.434,410.839,172.718,32.725,156.067
C00741=1060.315,219.682,410.812,172.720,32.729,156.068
C00742=1060.321,219.930,410.786,172.722,32.733,156.069
C00743=1060.327,220.179,410.761,172.724,32.737,156.069
C00744=1060.334,220.428,410.734,172.726,32.741,156.070
C00745=1060.340,220.676,410.707,172.729,32.745,156.071
C00746=1060.346,220.925,410.681,172.731,32.749,156.071
C00747=1060.352,221.158,410.657,172.733,32.752,156.072
C00748=1060.357,221.391,410.632,172.735,32.756,156.073
C00749=1060.363,221.624,410.607,172.737,32.760,156.074
C00750=1060.368,221.857,410.582,172.738,32.763,156.074
C00751=1060.374,222.089,410.557,172.740,32.767,156.075
C00752=1060.380,222.322,410.532,172.742,32.771,156.076
C00753=1060.386,222.555,410.507,172.743,32.774,156.076
C00754=1060.391,222.788,410.483,172.745,32.778,156.077
C00755=1060.397,223.036,410.456,172.747,32.782,156.078
C00756=1060.404,223.285,410.429,172.750,32.786,156.078
C00757=1060.410,223.533,410.403,172.752,32.790,156.079
C00758=1060.416,223.781,410.376,172.754,32.794,156.080
C00759=1060.422,224.030,410.350,172.756,32.798,156.081
C00760=1060.428,224.279,410.323,172.758,32.802,156.081
C00761=1060.434,224.527,410.296,172.760,32.805,156.082
C00762=1060.440,224.775,410.270,172.762,32.810,156.083
C00763=1060.447,225.024,410.243,172.764,32.813,156.084
C00764=1060.452,225.273,410.216,172.767,32.818,156.084
C00765=1060.458,225.521,410.190,172.769,32.821,156.085
C00766=1060.465,225.770,410.163,172.771,32.825,156.086
C00767=1060.471,226.018,410.137,172.773,32.829,156.087
C00768=1060.477,226.267,410.110,172.775,32.833,156.087
C00769=1060.483,226.516,410.083,172.777,32.837,156.088
C00770=1060.489,226.764,410.056,172.779,32.841,156.089
C00771=1060.495,227.013,410.029,172.782,32.845,156.089
C00772=1060.501,227.261,410.003,172.784,32.849,156.090
C00773=1060.508,227.509,409.977,172.786,32.853,156.091
C00774=1060.514,227.758,409.949,172.788,32.856,156.092
C00775=1060.520,228.006,409.922,172.790,32.861,156.092
C00776=1060.527,228.255,409.895,172.792,32.864,156.093
C00777=1060.532,228.504,409.869,172.795,32.868,156.094
C00778=1060.538,228.752,409.842,172.797,32.872,156.095
C00779=1060.544,229.001,409.815,172.799,32.876,156.095
C00780=1060.551,229.248,409.788,172.801,32.880,156.096
C00781=1060.558,229.498,409.761,172.803,32.883,156.097
C00782=1060.563,229.746,409.734,172.805,32.887,156.097
C00783=1060.570,229.995,409.707,172.808,32.891,156.098
C00784=1060.576,230.243,409.680,172.810,32.895,156.099
C00785=1060.582,230.491,409.653,172.812,32.899,156.100
C00786=1060.588,230.740,409.626,172.814,32.903,156.100
C00787=1060.594,230.988,409.599,172.816,32.907,156.101
C00788=1060.600,231.237,409.572,172.819,32.911,156.102
C00789=1060.606,231.486,409.545,172.821,32.915,156.103
C00790=1060.612,231.733,409.517,172.823,32.919,156.103
C00791=1060.618,231.982,409.490,172.825,32.922,156.104
C00792=1060.624,232.231,409.464,172.827,32.927,156.105
C00793=1060.630,232.479,409.436,172.830,32.930,156.105
C00794=1060.636,232.728,409.409,172.832,32.934,156.106
C00795=1060.643,232.977,409.382,172.834,32.938,156.107
C00796=1060.649,233.224,409.355,172.836,32.942,156.108
C00797=1060.655,233.473,409.328,172.838,32.945,156.108
C00798=1060.661,233.721,409.301,172.841,32.950,156.109
C00799=1060.667,233.971,409.273,172.843,32.953,156.110
C00800=1060.673,234.218,409.246,172.845,32.958,156.111
C00801=1060.679,234.467,409.219,172.847,32.961,156.111
C00802=1060.685,234.715,409.191,172.849,32.965,156.112
C00803=1060.691,234.944,409.166,172.851,32.969,156.113
C00804=1060.697,235.173,409.141,172.853,32.972,156.113
C00805=1060.703,235.402,409.116,172.856,32.976,156.114
C00806=1060.707,235.631,409.091,172.858,32.980,156.115
C00807=1060.713,235.860,409.065,172.860,32.983,156.115
C00808=1060.718,236.089,409.040,172.862,32.987,156.116
C00809=1060.725,236.318,409.015,172.864,32.990,156.117
C00810=1060.730,236.546,408.990,172.866,32.994,156.117
C00811=1060.736,236.795,408.963,172.868,32.998,156.118
C00812=1060.742,237.043,408.935,172.870,33.002,156.119
C00813=1060.748,237.292,408.907,172.873,33.005,156.119
C00814=1060.754,237.540,408.880,172.875,33.010,156.120
C00815=1060.761,237.789,408.853,172.877,33.013,156.121
C00816=1060.768,238.037,408.825,172.879,33.017,156.122
C00817=1060.773,238.286,408.798,172.882,33.021,156.122
C00818=1060.779,238.534,408.770,172.884,33.025,156.123
C00819=1060.785,238.782,408.743,172.886,33.029,156.124
C00820=1060.792,239.031,408.716,172.888,33.032,156.125
C00821=1060.798,239.280,408.687,172.891,33.037,156.125
C00822=1060.804,239.527,408.660,172.893,33.040,156.126
C00823=1060.810,239.776,408.632,172.895,33.044,156.127
C00824=1060.815,240.024,408.605,172.897,33.048,156.128
C00825=1060.822,240.273,408.577,172.900,33.052,156.128
C00826=1060.829,240.521,408.549,172.902,33.055,156.129
C00827=1060.835,240.769,408.522,172.904,33.059,156.130
C00828=1060.841,241.018,408.494,172.907,33.063,156.130
C00829=1060.847,241.267,408.467,172.909,33.067,156.131
C00830=1060.853,241.515,408.439,172.911,33.071,156.132
C00831=1060.859,241.763,408.411,172.913,33.075,156.133
C00832=1060.866,242.012,408.383,172.916,33.079,156.133
C00833=1060.872,242.260,408.356,172.918,33.082,156.134
C00834=1060.878,242.508,408.328,172.920,33.087,156.135
C00835=1060.884,242.757,408.299,172.923,33.090,156.135
C00836=1060.890,243.005,408.272,172.925,33.094,156.136
C00837=1060.896,243.254,408.244,172.927,33.098,156.137
C00838=1060.902,243.502,408.217,172.930,33.102,156.138
C00839=1060.908,243.751,408.189,172.932,33.105,156.138
C00840=1060.914,243.999,408.161,172.934,33.110,156.139
C00841=1060.920,244.247,408.133,172.936,33.113,156.140
C00842=1060.926,244.496,408.105,172.939,33.117,156.140
C00843=1060.932,244.744,408.077,172.941,33.121,156.141
C00844=1060.938,244.992,408.049,172.944,33.125,156.142
C00845=1060.944,245.241,408.021,172.947,33.129,156.143
C00846=1060.951,245.489,407.993,172.949,33.133,156.143
C00847=1060.957,245.737,407.964,172.951,33.137,156.144
C00848=1060.963,245.985,407.936,172.954,33.140,156.145
C00849=1060.969,246.234,407.909,172.956,33.144,156.146
C00850=1060.975,246.483,407.880,172.958,33.148,156.146
C00851=1060.981,246.731,407.852,172.961,33.152,156.147
C00852=1060.987,246.979,407.825,172.963,33.156,156.148
C00853=1060.993,247.228,407.796,172.965,33.160,156.149
C00854=1060.999,247.476,407.767,172.968,33.164,156.149
C00855=1061.005,247.724,407.739,172.970,33.168,156.150
C00856=1061.011,247.973,407.712,172.972,33.172,156.151
C00857=1061.017,248.221,407.683,172.975,33.176,156.152
C00858=1061.023,248.469,407.655,172.977,33.179,156.152
C00859=1061.028,248.695,407.629,172.979,33.183,156.153
C00860=1061.034,248.921,407.604,172.981,33.186,156.154
C00861=1061.040,249.147,407.577,172.983,33.190,156.154
C00862=1061.045,249.372,407.552,172.985,33.194,156.155
C00863=1061.050,249.598,407.527,172.988,33.197,156.156
C00864=1061.056,249.824,407.501,172.990,33.200,156.156
C00865=1061.061,250.050,407.475,172.992,33.204,156.157
C00866=1061.067,250.276,407.449,172.994,33.208,156.158
C00867=1061.073,250.524,407.421,172.996,33.211,156.158
C00868=1061.079,250.772,407.393,172.999,33.216,156.159
C00869=1061.085,251.020,407.364,173.001,33.219,156.160
C00870=1061.091,251.269,407.335,173.004,33.223,156.161
C00871=1061.097,251.517,407.306,173.006,33.227,156.161
C00872=1061.104,251.766,407.279,173.008,33.231,156.162
C00873=1061.109,252.014,407.251,173.011,33.235,156.163
C00874=1061.115,252.262,407.222,173.013,33.239,156.164
C00875=1061.121,252.511,407.193,173.015,33.242,156.164
C00876=1061.128,252.759,407.164,173.018,33.247,156.165
C00877=1061.134,253.008,407.136,173.021,33.250,156.166
C00878=1061.141,253.255,407.107,173.024,33.254,156.166
C00879=1061.146,253.503,407.079,173.026,33.258,156.167
C00880=1061.152,253.752,407.050,173.028,33.262,156.168
C00881=1061.158,254.000,407.022,173.031,33.266,156.169
C00882=1061.164,254.249,406.993,173.033,33.270,156.169
C00883=1061.170,254.497,406.965,173.036,33.273,156.170
C00884=1061.177,254.745,406.936,173.038,33.277,156.171
C00885=1061.183,254.994,406.908,173.040,33.281,156.172
C00886=1061.189,255.242,406.879,173.043,33.285,156.172
C00887=1061.195,255.489,406.850,173.045,33.289,156.173
C00888=1061.201,255.738,406.822,173.048,33.292,156.174
C00889=1061.207,255.986,406.793,173.050,33.297,156.175
C00890=1061.213,256.235,406.765,173.053,33.300,156.175
C00891=1061.219,256.483,406.736,173.055,33.304,156.176
C00892=1061.226,256.731,406.707,173.057,33.308,156.177
C00893=1061.232,256.980,406.679,173.060,33.312,156.177
C00894=1061.239,257.228,406.650,173.062,33.315,156.178
C00895=1061.245,257.476,406.621,173.065,33.319,156.179
C00896=1061.251,257.725,406.592,173.067,33.323,156.180
C00897=1061.257,257.973,406.563,173.070,33.327,156.180
C00898=1061.263,258.221,406.534,173.072,33.331,156.181
C00899=1061.270,258.469,406.505,173.076,33.335,156.182
C00900=1061.276,258.718,406.477,173.078,33.338,156.183
C00901=1061.282,258.966,406.448,173.081,33.342,156.183
C00902=1061.288,259.214,406.419,173.083,33.346,156.184
C00903=1061.294,259.462,406.390,173.085,33.350,156.185
C00904=1061.300,259.711,406.361,173.088,33.354,156.185
C00905=1061.307,259.959,406.333,173.090,33.357,156.186
C00906=1061.313,260.207,406.304,173.093,33.361,156.187
C00907=1061.320,260.455,406.275,173.095,33.365,156.188
C00908=1061.326,260.703,406.246,173.098,33.369,156.188
C00909=1061.332,260.951,406.217,173.100,33.373,156.189
C00910=1061.338,261.200,406.188,173.103,33.376,156.190
C00911=1061.345,261.449,406.159,173.105,33.380,156.190
C00912=1061.351,261.697,406.130,173.108,33.384,156.191
C00913=1061.358,261.945,406.101,173.110,33.388,156.192
C00914=1061.364,262.193,406.072,173.113,33.391,156.193
C00915=1061.370,262.418,406.046,173.115,33.395,156.193
C00916=1061.375,262.643,406.019,173.117,33.399,156.194
C00917=1061.381,262.867,405.993,173.120,33.402,156.195
C00918=1061.387,263.092,405.967,173.123,33.405,156.195
C00919=1061.392,263.317,405.940,173.125,33.408,156.196
C00920=1061.398,263.541,405.914,173.128,33.412,156.197
C00921=1061.403,263.766,405.888,173.130,33.416,156.197
C00922=1061.409,263.991,405.861,173.132,33.419,156.198
C00923=1061.415,264.239,405.832,173.135,33.423,156.199
C00924=1061.421,264.487,405.803,173.137,33.427,156.199
C00925=1061.428,264.735,405.774,173.140,33.431,156.200
C00926=1061.433,264.984,405.744,173.142,33.434,156.201
C00927=1061.439,265.232,405.715,173.145,33.439,156.202
C00928=1061.446,265.480,405.685,173.147,33.442,156.202
C00929=1061.452,265.729,405.655,173.150,33.447,156.203
C00930=1061.458,265.977,405.626,173.152,33.450,156.204
C00931=1061.464,266.225,405.597,173.155,33.454,156.205
C00932=1061.470,266.473,405.567,173.157,33.458,156.205
C00933=1061.477,266.721,405.538,173.160,33.462,156.206
C00934=1061.483,266.969,405.509,173.163,33.465,156.207
C00935=1061.489,267.217,405.480,173.166,33.470,156.208
C00936=1061.495,267.466,405.450,173.168,33.473,156.208
C00937=1061.502,267.714,405.420,173.171,33.477,156.209
C00938=1061.508,267.962,405.391,173.174,33.481,156.210
C00939=1061.513,268.210,405.361,173.176,33.485,156.210
C00940=1061.520,268.459,405.332,173.179,33.489,156.211
C00941=1061.527,268.707,405.302,173.181,33.493,156.212
C00942=1061.532,268.955,405.272,173.184,33.496,156.213
C00943=1061.539,269.203,405.243,173.186,33.500,156.213
C00944=1061.544,269.451,405.213,173.189,33.504,156.214
C00945=1061.551,269.699,405.184,173.191,33.508,156.215
C00946=1061.557,269.947,405.154,173.194,33.512,156.216
C00947=1061.563,270.196,405.124,173.197,33.516,156.216
C00948=1061.570,270.443,405.094,173.200,33.520,156.217
C00949=1061.575,270.692,405.065,173.203,33.524,156.218
C00950=1061.582,270.940,405.036,173.205,33.528,156.219
C00951=1061.588,271.188,405.005,173.208,33.531,156.219
C00952=1061.594,271.437,404.976,173.210,33.536,156.220
C00953=1061.600,271.685,404.946,173.213,33.539,156.221
C00954=1061.606,271.933,404.917,173.216,33.543,156.222
C00955=1061.612,272.180,404.886,173.218,33.547,156.222
C00956=1061.619,272.429,404.857,173.221,33.551,156.223
C00957=1061.625,272.677,404.826,173.223,33.555,156.224
C00958=1061.631,272.925,404.797,173.226,33.559,156.225
C00959=1061.638,273.174,404.767,173.229,33.563,156.225
C00960=1061.643,273.422,404.736,173.232,33.566,156.226
C00961=1061.650,273.670,404.707,173.235,33.570,156.227
C00962=1061.655,273.918,404.677,173.237,33.574,156.228
C00963=1061.663,274.166,404.647,173.240,33.578,156.228
C00964=1061.668,274.414,404.617,173.243,33.582,156.229
C00965=1061.674,274.662,404.587,173.245,33.586,156.230
C00966=1061.681,274.910,404.557,173.248,33.590,156.231
C00967=1061.687,275.158,404.526,173.251,33.594,156.231
C00968=1061.692,275.407,404.497,173.253,33.598,156.232
C00969=1061.699,275.654,404.467,173.256,33.601,156.233
C00970=1061.705,275.903,404.436,173.258,33.606,156.234
C00971=1061.710,276.129,404.409,173.261,33.609,156.234
C00972=1061.717,276.356,404.382,173.264,33.612,156.235
C00973=1061.722,276.583,404.354,173.267,33.616,156.236
C00974=1061.728,276.809,404.326,173.269,33.620,156.236
C00975=1061.734,277.036,404.299,173.271,33.623,156.237
C00976=1061.738,277.262,404.271,173.274,33.627,156.238
C00977=1061.745,277.488,404.244,173.276,33.630,156.239
C00978=1061.751,277.715,404.216,173.279,33.634,156.239
C00979=1061.756,277.963,404.186,173.281,33.638,156.240
C00980=1061.763,278.212,404.155,173.284,33.642,156.241
C00981=1061.769,278.459,404.125,173.287,33.646,156.241
C00982=1061.775,278.708,404.096,173.289,33.650,156.242
C00983=1061.781,278.956,404.065,173.293,33.653,156.243
C00984=1061.787,279.204,404.035,173.296,33.658,156.244
C00985=1061.794,279.452,404.004,173.298,33.661,156.245
C00986=1061.800,279.700,403.974,173.301,33.665,156.245
C00987=1061.806,279.948,403.943,173.304,33.669,156.246
C00988=1061.812,280.196,403.913,173.306,33.673,156.247
C00989=1061.818,280.444,403.883,173.309,33.677,156.248
C00990=1061.825,280.693,403.852,173.312,33.681,156.248
C00991=1061.830,280.940,403.822,173.314,33.685,156.249
C00992=1061.837,281.189,403.791,173.317,33.689,156.250
C00993=1061.844,281.436,403.760,173.321,33.693,156.251
C00994=1061.849,281.684,403.730,173.323,33.697,156.251
C00995=1061.856,281.932,403.699,173.326,33.701,156.252
C00996=1061.862,282.180,403.669,173.329,33.705,156.253
C00997=1061.868,282.429,403.638,173.331,33.709,156.254
C00998=1061.874,282.676,403.608,173.334,33.713,156.255
C00999=1061.880,282.925,403.577,173.337,33.717,156.255
C01000=1061.886,283.172,403.546,173.340,33.721,156.256
C01001=1061.893,283.421,403.515,173.342,33.725,156.257
C01002=1061.899,283.668,403.485,173.345,33.729,156.258
C01003=1061.905,283.917,403.454,173.349,33.733,156.258
C01004=1061.911,284.164,403.423,173.351,33.736,156.259
C01005=1061.918,284.413,403.393,173.354,33.741,156.260
C01006=1061.923,284.661,403.362,173.357,33.745,156.261
C01007=1061.930,284.909,403.331,173.360,33.748,156.262
C01008=1061.936,285.156,403.300,173.362,33.753,156.262
C01009=1061.942,285.405,403.270,173.365,33.756,156.263
C01010=1061.948,285.653,403.239,173.368,33.760,156.264
C01011=1061.955,285.900,403.208,173.372,33.765,156.265
C01012=1061.961,286.148,403.178,173.374,33.768,156.265
C01013=1061.968,286.396,403.146,173.377,33.772,156.266
C01014=1061.973,286.644,403.116,173.380,33.776,156.267
C01015=1061.980,286.893,403.085,173.383,33.780,156.268
C01016=1061.986,287.140,403.054,173.385,33.784,156.268
C01017=1061.992,287.388,403.023,173.388,33.788,156.269
C01018=1061.999,287.636,402.992,173.391,33.792,156.270
C01019=1062.005,287.884,402.961,173.394,33.796,156.271
C01020=1062.012,288.132,402.930,173.397,33.800,156.272
C01021=1062.017,288.381,402.899,173.400,33.804,156.272
C01022=1062.023,288.628,402.868,173.403,33.808,156.273
C01023=1062.030,288.876,402.837,173.406,33.812,156.274
C01024=1062.036,289.124,402.806,173.408,33.816,156.275
C01025=1062.042,289.372,402.775,173.411,33.820,156.276
C01026=1062.048,289.620,402.743,173.414,33.824,156.276
C01027=1062.054,289.852,402.714,173.417,33.828,156.277
C01028=1062.060,290.084,402.686,173.420,33.831,156.278
C01029=1062.066,290.316,402.657,173.423,33.835,156.279
C01030=1062.072,290.548,402.627,173.425,33.839,156.279
C01031=1062.078,290.779,402.597,173.428,33.843,156.280
C01032=1062.083,291.011,402.569,173.431,33.846,156.281
C01033=1062.089,291.244,402.539,173.433,33.850,156.282
C01034=1062.095,291.476,402.510,173.436,33.854,156.282
C01035=1062.102,291.724,402.479,173.439,33.858,156.283
C01036=1062.108,291.971,402.448,173.443,33.862,156.284
C01037=1062.114,292.220,402.416,173.445,33.866,156.285
C01038=1062.120,292.468,402.385,173.448,33.870,156.285
C01039=1062.126,292.715,402.354,173.451,33.874,156.286
C01040=1062.132,292.963,402.322,173.454,33.879,156.287
C01041=1062.139,293.211,402.291,173.457,33.882,156.288
C01042=1062.145,293.459,402.260,173.459,33.886,156.289
C01043=1062.151,293.707,402.228,173.462,33.890,156.289
C01044=1062.158,293.955,402.196,173.466,33.895,156.290
C01045=1062.164,294.203,402.165,173.469,33.898,156.291
C01046=1062.170,294.450,402.133,173.472,33.902,156.292
C01047=1062.176,294.698,402.102,173.475,33.907,156.293
C01048=1062.183,294.947,402.071,173.477,33.911,156.294
C01049=1062.189,295.195,402.039,173.480,33.914,156.294
C01050=1062.195,295.442,402.008,173.483,33.919,156.295
C01051=1062.201,295.690,401.976,173.487,33.923,156.296
C01052=1062.208,295.938,401.945,173.490,33.927,156.297
C01053=1062.214,296.186,401.913,173.493,33.931,156.298
C01054=1062.220,296.434,401.882,173.496,33.935,156.298
C01055=1062.226,296.682,401.849,173.498,33.939,156.299
C01056=1062.233,296.930,401.818,173.501,33.943,156.300
C01057=1062.239,297.177,401.785,173.504,33.947,156.301
C01058=1062.246,297.425,401.754,173.508,33.951,156.302
C01059=1062.251,297.673,401.722,173.511,33.956,156.302
C01060=1062.257,297.921,401.690,173.514,33.960,156.303
C01061=1062.263,298.169,401.658,173.517,33.964,156.304
C01062=1062.270,298.417,401.627,173.519,33.968,156.305
C01063=1062.275,298.664,401.594,173.522,33.972,156.306
C01064=1062.281,298.912,401.562,173.525,33.976,156.307
C01065=1062.287,299.160,401.530,173.529,33.981,156.307
C01066=1062.294,299.408,401.499,173.532,33.985,156.308
C01067=1062.300,299.655,401.466,173.535,33.989,156.309
C01068=1062.306,299.903,401.434,173.538,33.993,156.310
C01069=1062.312,300.152,401.402,173.541,33.997,156.311
C01070=1062.318,300.399,401.371,173.543,34.001,156.312
C01071=1062.325,300.647,401.338,173.547,34.006,156.312
C01072=1062.330,300.895,401.307,173.550,34.010,156.313
C01073=1062.336,301.143,401.275,173.553,34.014,156.314
C01074=1062.343,301.390,401.242,173.556,34.018,156.315
C01075=1062.349,301.638,401.210,173.559,34.022,156.316
C01076=1062.355,301.886,401.178,173.562,34.026,156.317
C01077=1062.361,302.134,401.146,173.566,34.031,156.317
C01078=1062.368,302.382,401.114,173.569,34.035,156.318
C01079=1062.374,302.630,401.081,173.572,34.039,156.319
C01080=1062.380,302.877,401.050,173.575,34.043,156.320
C01081=1062.386,303.125,401.017,173.578,34.047,156.321
C01082=1062.392,303.373,400.985,173.581,34.051,156.322
C01083=1062.399,303.612,400.954,173.584,34.056,156.322
C01084=1062.404,303.852,400.923,173.587,34.060,156.323
C01085=1062.411,304.091,400.891,173.590,34.064,156.324
C01086=1062.417,304.330,400.860,173.593,34.068,156.325
C01087=1062.423,304.570,400.829,173.596,34.072,156.326
C01088=1062.429,304.810,400.797,173.599,34.076,156.326
C01089=1062.434,305.050,400.767,173.603,34.080,156.327
C01090=1062.441,305.289,400.736,173.605,34.084,156.328
C01091=1062.448,305.537,400.703,173.608,34.088,156.329
C01092=1062.454,305.785,400.670,173.611,34.092,156.330
C01093=1062.460,306.033,400.638,173.614,34.097,156.331
C01094=1062.466,306.280,400.605,173.617,34.101,156.331
C01095=1062.472,306.528,400.573,173.621,34.105,156.332
C01096=1062.479,306.776,400.541,173.624,34.109,156.333
C01097=1062.486,307.023,400.508,173.627,34.114,156.334
C01098=1062.492,307.271,400.476,173.630,34.118,156.335
C01099=1062.498,307.519,400.443,173.633,34.122,156.336
C01100=1062.504,307.767,400.411,173.636,34.126,156.337
C01101=1062.510,308.014,400.378,173.640,34.130,156.337
C01102=1062.517,308.262,400.345,173.643,34.135,156.338
C01103=1062.524,308.510,400.312,173.646,34.139,156.339
C01104=1062.530,308.758,400.281,173.649,34.143,156.340
C01105=1062.537,309.006,400.248,173.652,34.147,156.341
C01106=1062.543,309.253,400.215,173.656,34.152,156.342
C01107=1062.549,309.501,400.183,173.659,34.156,156.343
C01108=1062.555,309.749,400.150,173.662,34.160,156.343
C01109=1062.562,309.996,400.117,173.665,34.164,156.344
C01110=1062.569,310.244,400.084,173.669,34.168,156.345
C01111=1062.575,310.492,400.051,173.673,34.172,156.346
C01112=1062.581,310.740,400.019,173.676,34.177,156.347
C01113=1062.588,310.988,399.987,173.679,34.181,156.348
C01114=1062.594,311.235,399.954,173.682,34.185,156.349
C01115=1062.601,311.483,399.921,173.685,34.190,156.349
C01116=1062.607,311.731,399.889,173.688,34.194,156.350
C01117=1062.614,311.979,399.856,173.692,34.198,156.351
C01118=1062.620,312.226,399.823,173.695,34.202,156.352
C01119=1062.627,312.473,399.790,173.698,34.206,156.353
C01120=1062.634,312.722,399.757,173.701,34.211,156.354
C01121=1062.640,312.969,399.724,173.704,34.215,156.355
C01122=1062.646,313.217,399.691,173.708,34.219,156.355
C01123=1062.653,313.465,399.658,173.711,34.223,156.356
C01124=1062.659,313.713,399.625,173.714,34.227,156.357
C01125=1062.666,313.960,399.592,173.718,34.232,156.358
C01126=1062.672,314.208,399.560,173.721,34.236,156.359
C01127=1062.678,314.456,399.525,173.725,34.241,156.360
C01128=1062.685,314.703,399.493,173.728,34.245,156.361
C01129=1062.690,314.951,399.459,173.731,34.250,156.362
C01130=1062.696,315.199,399.426,173.734,34.254,156.362
C01131=1062.702,315.446,399.392,173.738,34.259,156.363
C01132=1062.709,315.694,399.359,173.741,34.263,156.364
C01133=1062.716,315.942,399.327,173.744,34.268,156.365
C01134=1062.721,316.189,399.293,173.747,34.272,156.366
C01135=1062.728,316.437,399.260,173.750,34.276,156.367
C01136=1062.734,316.685,399.225,173.754,34.280,156.368
C01137=1062.740,316.932,399.193,173.757,34.285,156.369
C01138=1062.746,317.180,399.159,173.760,34.290,156.370
C01139=1062.753,317.422,399.126,173.763,34.294,156.371
C01140=1062.759,317.663,399.094,173.766,34.298,156.371
C01141=1062.765,317.905,399.062,173.770,34.303,156.372
C01142=1062.771,318.146,399.029,173.774,34.307,156.373
C01143=1062.777,318.387,398.996,173.777,34.311,156.374
C01144=1062.783,318.629,398.963,173.780,34.316,156.375
C01145=1062.789,318.870,398.930,173.784,34.320,156.376
C01146=1062.795,319.112,398.898,173.787,34.325,156.377
C01147=1062.802,319.359,398.865,173.790,34.329,156.378
C01148=1062.808,319.608,398.831,173.793,34.333,156.379
C01149=1062.814,319.854,398.797,173.796,34.338,156.380
C01150=1062.821,320.102,398.763,173.800,34.342,156.381
C01151=1062.827,320.350,398.730,173.803,34.347,156.381
C01152=1062.833,320.597,398.696,173.806,34.351,156.382
C01153=1062.840,320.845,398.662,173.810,34.356,156.383
C01154=1062.846,321.093,398.629,173.814,34.360,156.384
C01155=1062.853,321.341,398.595,173.817,34.365,156.385
C01156=1062.859,321.588,398.561,173.820,34.369,156.386
C01157=1062.865,321.836,398.527,173.823,34.374,156.387
C01158=1062.872,322.083,398.494,173.827,34.378,156.388
C01159=1062.877,322.331,398.460,173.831,34.383,156.389
C01160=1062.885,322.578,398.426,173.834,34.387,156.390
C01161=1062.890,322.826,398.393,173.837,34.392,156.391
C01162=1062.897,323.074,398.359,173.841,34.396,156.392
C01163=1062.903,323.321,398.325,173.844,34.401,156.393
C01164=1062.911,323.569,398.291,173.848,34.405,156.393
C01165=1062.917,323.817,398.257,173.851,34.410,156.394
C01166=1062.923,324.064,398.223,173.855,34.414,156.395
C01167=1062.930,324.313,398.189,173.858,34.419,156.396
C01168=1062.936,324.560,398.155,173.861,34.423,156.397
C01169=1062.943,324.807,398.122,173.865,34.428,156.398
C01170=1062.949,325.055,398.088,173.869,34.433,156.399
C01171=1062.955,325.303,398.053,173.872,34.437,156.400
C01172=1062.962,325.550,398.019,173.875,34.441,156.401
C01173=1062.968,325.798,397.985,173.878,34.446,156.402
C01174=1062.975,326.045,397.951,173.883,34.451,156.403
C01175=1062.981,326.293,397.917,173.886,34.455,156.404
C01176=1062.988,326.541,397.883,173.889,34.459,156.405
C01177=1062.995,326.788,397.849,173.892,34.464,156.406
C01178=1063.001,327.036,397.815,173.897,34.469,156.407
C01179=1063.008,327.283,397.781,173.900,34.473,156.408
C01180=1063.015,327.531,397.746,173.903,34.478,156.409
C01181=1063.021,327.778,397.712,173.906,34.483,156.410
C01182=1063.028,328.026,397.678,173.911,34.487,156.410
C01183=1063.034,328.274,397.644,173.914,34.492,156.411
C01184=1063.041,328.522,397.609,173.917,34.496,156.412
C01185=1063.047,328.769,397.576,173.921,34.501,156.413
C01186=1063.054,329.017,397.542,173.925,34.506,156.414
C01187=1063.061,329.264,397.506,173.928,34.510,156.415
C01188=1063.068,329.512,397.473,173.931,34.515,156.416
C01189=1063.074,329.759,397.439,173.936,34.520,156.417
C01190=1063.080,330.007,397.404,173.939,34.524,156.418
C01191=1063.088,330.254,397.370,173.942,34.528,156.419
C01192=1063.094,330.502,397.335,173.946,34.533,156.420
C01193=1063.100,330.750,397.301,173.950,34.538,156.421
C01194=1063.107,330.997,397.266,173.953,34.542,156.422
C01195=1063.113,331.228,397.233,173.956,34.547,156.423
C01196=1063.119,331.459,397.202,173.959,34.552,156.424
C01197=1063.125,331.690,397.169,173.964,34.556,156.425
C01198=1063.131,331.922,397.137,173.967,34.560,156.426
C01199=1063.136,332.153,397.105,173.970,34.564,156.427
C01200=1063.142,332.384,397.072,173.973,34.569,156.428
C01201=1063.149,332.615,397.040,173.977,34.574,156.429
C01202=1063.155,332.845,397.007,173.980,34.578,156.429
C01203=1063.162,333.093,396.973,173.983,34.583,156.431
C01204=1063.168,333.341,396.937,173.988,34.588,156.432
C01205=1063.175,333.589,396.903,173.991,34.592,156.433
C01206=1063.181,333.835,396.868,173.994,34.597,156.433
C01207=1063.187,334.083,396.834,173.999,34.602,156.435
C01208=1063.194,334.331,396.799,174.002,34.607,156.436
C01209=1063.200,334.578,396.763,174.005,34.611,156.437
C01210=1063.207,334.826,396.729,174.009,34.616,156.438
C01211=1063.213,335.074,396.693,174.013,34.621,156.439
C01212=1063.220,335.321,396.658,174.016,34.626,156.440
C01213=1063.226,335.568,396.624,174.020,34.631,156.441
C01214=1063.233,335.816,396.589,174.024,34.636,156.442
C01215=1063.240,336.063,396.554,174.028,34.641,156.443
C01216=1063.246,336.311,396.519,174.031,34.645,156.444
C01217=1063.253,336.558,396.484,174.035,34.650,156.445
C01218=1063.260,336.806,396.449,174.039,34.655,156.446
C01219=1063.267,337.068,396.411,174.042,34.660,156.447
C01220=1063.273,337.330,396.374,174.047,34.665,156.448
C01221=1063.280,337.592,396.337,174.050,34.671,156.449
C01222=1063.287,337.855,396.300,174.054,34.676,156.450
C01223=1063.294,338.103,396.265,174.058,34.680,156.451
C01224=1063.301,338.350,396.229,174.062,34.686,156.452
C01225=1063.307,338.598,396.194,174.065,34.690,156.453
C01226=1063.313,338.845,396.159,174.070,34.696,156.454
C01227=1063.320,339.092,396.123,174.073,34.701,156.455
C01228=1063.326,339.340,396.088,174.076,34.705,156.456
C01229=1063.333,339.587,396.053,174.081,34.711,156.458
C01230=1063.340,339.835,396.017,174.084,34.715,156.458
C01231=1063.346,340.082,395.982,174.088,34.720,156.460
C01232=1063.352,340.330,395.947,174.092,34.725,156.461
C01233=1063.360,340.576,395.911,174.096,34.730,156.462
C01234=1063.366,340.824,395.876,174.099,34.735,156.463
C01235=1063.372,341.072,395.840,174.104,34.740,156.464
C01236=1063.379,341.319,395.805,174.107,34.745,156.465
C01237=1063.385,341.567,395.769,174.110,34.750,156.466
C01238=1063.392,341.814,395.734,174.115,34.755,156.467
C01239=1063.399,342.061,395.698,174.118,34.760,156.468
C01240=1063.405,342.308,395.662,174.122,34.765,156.469
C01241=1063.412,342.556,395.627,174.126,34.771,156.470
C01242=1063.419,342.802,395.591,174.130,34.775,156.471
C01243=1063.425,343.050,395.556,174.133,34.780,156.472
C01244=1063.432,343.298,395.520,174.138,34.786,156.474
C01245=1063.439,343.546,395.485,174.141,34.790,156.475
C01246=1063.445,343.793,395.449,174.145,34.795,156.476
C01247=1063.451,344.040,395.413,174.149,34.800,156.477
C01248=1063.458,344.287,395.377,174.153,34.806,156.478
C01249=1063.465,344.535,395.341,174.157,34.811,156.479
C01250=1063.472,344.781,395.305,174.161,34.816,156.480
C01251=1063.478,345.018,395.271,174.164,34.821,156.481
C01252=1063.484,345.254,395.237,174.168,34.826,156.482
C01253=1063.491,345.491,395.203,174.172,34.831,156.483
C01254=1063.496,345.727,395.168,174.175,34.836,156.484
C01255=1063.503,345.963,395.134,174.180,34.841,156.485
C01256=1063.509,346.199,395.100,174.183,34.845,156.486
C01257=1063.516,346.435,395.064,174.186,34.850,156.487
C01258=1063.522,346.671,395.031,174.191,34.856,156.489
C01259=1063.528,346.918,394.994,174.194,34.861,156.490
C01260=1063.536,347.167,394.959,174.199,34.866,156.491
C01261=1063.542,347.414,394.922,174.202,34.871,156.492
C01262=1063.549,347.660,394.886,174.206,34.876,156.493
C01263=1063.555,347.908,394.851,174.210,34.881,156.494
C01264=1063.561,348.155,394.814,174.214,34.887,156.495
C01265=1063.568,348.403,394.777,174.218,34.892,156.496
C01266=1063.575,348.650,394.742,174.222,34.898,156.498
C01267=1063.582,348.897,394.705,174.226,34.903,156.499
C01268=1063.588,349.145,394.669,174.230,34.908,156.500
C01269=1063.595,349.392,394.633,174.234,34.913,156.501
C01270=1063.602,349.639,394.597,174.237,34.918,156.502
C01271=1063.609,349.887,394.560,174.242,34.924,156.503
C01272=1063.615,350.134,394.524,174.246,34.929,156.504
C01273=1063.622,350.380,394.488,174.250,34.934,156.506
C01274=1063.629,350.628,394.451,174.254,34.939,156.507
C01275=1063.635,350.875,394.414,174.257,34.945,156.508
C01276=1063.642,351.122,394.378,174.262,34.950,156.509
C01277=1063.649,351.370,394.342,174.266,34.955,156.510
C01278=1063.656,351.617,394.305,174.270,34.961,156.511
C01279=1063.662,351.864,394.269,174.274,34.966,156.513
C01280=1063.669,352.112,394.232,174.279,34.971,156.514
C01281=1063.675,352.359,394.196,174.282,34.977,156.515
C01282=1063.682,352.606,394.159,174.286,34.982,156.516
C01283=1063.689,352.853,394.122,174.290,34.988,156.517
C01284=1063.696,353.100,394.087,174.294,34.993,156.518
C01285=1063.703,353.347,394.049,174.299,34.999,156.520
C01286=1063.709,353.594,394.013,174.302,35.004,156.521
C01287=1063.716,353.842,393.976,174.307,35.010,156.522
C01288=1063.722,354.089,393.939,174.311,35.015,156.523
C01289=1063.729,354.336,393.902,174.314,35.020,156.524
C01290=1063.736,354.583,393.865,174.319,35.026,156.526
C01291=1063.742,354.830,393.829,174.323,35.032,156.527
C01292=1063.749,355.078,393.792,174.327,35.037,156.528
C01293=1063.756,355.325,393.755,174.331,35.043,156.529
C01294=1063.763,355.572,393.718,174.336,35.048,156.530
C01295=1063.770,355.819,393.681,174.339,35.053,156.532
C01296=1063.776,356.067,393.644,174.344,35.059,156.533
C01297=1063.783,356.314,393.608,174.348,35.065,156.534
C01298=1063.790,356.561,393.570,174.352,35.070,156.535
C01299=1063.797,356.808,393.533,174.356,35.076,156.536
C01300=1063.804,357.055,393.496,174.360,35.081,156.538
C01301=1063.811,357.303,393.459,174.365,35.087,156.539
C01302=1063.817,357.549,393.422,174.368,35.093,156.540
C01303=1063.824,357.797,393.384,174.373,35.098,156.541
C01304=1063.830,358.044,393.348,174.377,35.103,156.543
C01305=1063.837,358.291,393.310,174.382,35.109,156.544
C01306=1063.844,358.538,393.273,174.385,35.115,156.545
C01307=1063.851,358.776,393.238,174.390,35.120,156.546
C01308=1063.858,359.014,393.201,174.394,35.126,156.548
C01309=1063.864,359.253,393.165,174.398,35.131,156.549
C01310=1063.870,359.491,393.130,174.402,35.137,156.550
C01311=1063.877,359.730,393.094,174.406,35.142,156.551
C01312=1063.884,359.967,393.058,174.410,35.148,156.552
C01313=1063.891,360.206,393.022,174.415,35.153,156.554
C01314=1063.897,360.444,392.986,174.418,35.159,156.555
C01315=1063.904,360.691,392.948,174.422,35.165,156.556
C01316=1063.910,360.939,392.910,174.427,35.170,156.557
C01317=1063.917,361.185,392.873,174.431,35.176,156.559
C01318=1063.924,361.432,392.836,174.435,35.182,156.560
C01319=1063.931,361.679,392.798,174.439,35.187,156.561
C01320=1063.937,361.926,392.760,174.444,35.194,156.563
C01321=1063.945,362.173,392.723,174.449,35.199,156.564
C01322=1063.952,362.420,392.685,174.453,35.205,156.565
C01323=1063.959,362.667,392.648,174.457,35.211,156.566
C01324=1063.965,362.914,392.610,174.461,35.217,156.568
C01325=1063.972,363.161,392.572,174.466,35.222,156.569
C01326=1063.979,363.408,392.535,174.470,35.228,156.570
C01327=1063.986,363.656,392.497,174.475,35.234,156.572
C01328=1063.993,363.903,392.459,174.479,35.240,156.573
C01329=1064.000,364.149,392.422,174.483,35.246,156.574
C01330=1064.006,364.397,392.384,174.487,35.252,156.576
C01331=1064.014,364.643,392.346,174.492,35.258,156.577
C01332=1064.020,364.891,392.308,174.496,35.264,156.578
C01333=1064.028,365.138,392.270,174.501,35.270,156.580
C01334=1064.034,365.385,392.232,174.505,35.275,156.581
C01335=1064.041,365.631,392.194,174.509,35.282,156.582
C01336=1064.048,365.879,392.156,174.514,35.288,156.584
C01337=1064.054,366.126,392.118,174.518,35.293,156.585
C01338=1064.062,366.373,392.080,174.523,35.300,156.586
C01339=1064.068,366.619,392.042,174.527,35.306,156.588
C01340=1064.075,366.866,392.004,174.532,35.311,156.589
C01341=1064.082,367.113,391.965,174.536,35.318,156.590
C01342=1064.089,367.361,391.928,174.541,35.324,156.592
C01343=1064.096,367.607,391.889,174.544,35.330,156.593
C01344=1064.102,367.855,391.851,174.549,35.336,156.594
C01345=1064.110,368.101,391.813,174.554,35.342,156.596
C01346=1064.116,368.349,391.775,174.558,35.348,156.597
C01347=1064.124,368.595,391.736,174.563,35.354,156.599
C01348=1064.131,368.842,391.697,174.567,35.360,156.600
C01349=1064.137,369.090,391.659,174.572,35.366,156.601
C01350=1064.145,369.336,391.621,174.576,35.373,156.603
C01351=1064.151,369.583,391.582,174.581,35.379,156.604
C01352=1064.159,369.830,391.545,174.586,35.385,156.606
C01353=1064.166,370.077,391.506,174.590,35.391,156.607
C01354=1064.172,370.324,391.467,174.595,35.397,156.608
C01355=1064.180,370.571,391.430,174.599,35.404,156.610
C01356=1064.186,370.818,391.391,174.604,35.410,156.611
C01357=1064.193,371.064,391.352,174.609,35.416,156.612
C01358=1064.201,371.311,391.314,174.613,35.422,156.614
C01359=1064.208,371.558,391.275,174.618,35.428,156.615
C01360=1064.215,371.804,391.237,174.622,35.434,156.617
C01361=1064.222,372.052,391.198,174.627,35.441,156.618
C01362=1064.228,372.299,391.160,174.632,35.447,156.620
C01363=1064.236,372.546,391.120,174.636,35.453,156.621
C01364=1064.243,372.793,391.082,174.641,35.460,156.622
C01365=1064.250,373.040,391.042,174.646,35.466,156.624
C01366=1064.257,373.288,391.004,174.650,35.472,156.625
C01367=1064.264,373.534,390.965,174.655,35.479,156.627
C01368=1064.270,373.781,390.926,174.660,35.485,156.628
C01369=1064.277,374.028,390.887,174.664,35.492,156.630
C01370=1064.284,374.275,390.848,174.669,35.498,156.631
C01371=1064.292,374.522,390.810,174.674,35.505,156.633
C01372=1064.299,374.769,390.771,174.678,35.511,156.634
C01373=1064.306,375.015,390.732,174.683,35.518,156.636
C01374=1064.313,375.262,390.692,174.688,35.524,156.637
C01375=1064.320,375.508,390.653,174.692,35.530,156.639
C01376=1064.327,375.755,390.615,174.697,35.537,156.640
C01377=1064.334,376.002,390.575,174.702,35.544,156.642
C01378=1064.341,376.249,390.536,174.706,35.550,156.643
C01379=1064.348,376.496,390.497,174.711,35.557,156.645
C01380=1064.355,376.742,390.458,174.716,35.563,156.646
C01381=1064.363,376.990,390.418,174.720,35.570,156.648
C01382=1064.369,377.236,390.379,174.726,35.576,156.649
C01383=1064.376,377.483,390.340,174.731,35.583,156.651
C01384=1064.383,377.729,390.301,174.735,35.589,156.652
C01385=1064.391,377.976,390.261,174.740,35.596,156.654
C01386=1064.398,378.223,390.222,174.745,35.603,156.655
C01387=1064.405,378.469,390.183,174.749,35.609,156.657
C01388=1064.413,378.716,390.143,174.754,35.616,156.658
C01389=1064.419,378.963,390.104,174.759,35.623,156.660
C01390=1064.427,379.210,390.064,174.765,35.629,156.661
C01391=1064.434,379.457,390.025,174.769,35.636,156.663
C01392=1064.441,379.703,389.986,174.774,35.643,156.664
C01393=1064.449,379.950,389.946,174.779,35.649,156.666
C01394=1064.456,380.197,389.907,174.783,35.656,156.668
C01395=1064.463,380.444,389.866,174.788,35.663,156.669
C01396=1064.470,380.690,389.827,174.794,35.670,156.671
C01397=1064.477,380.937,389.787,174.799,35.677,156.672
C01398=1064.484,381.184,389.748,174.803,35.683,156.674
C01399=1064.491,381.430,389.709,174.808,35.690,156.675
C01400=1064.498,381.677,389.668,174.813,35.697,156.677
C01401=1064.505,381.924,389.629,174.818,35.704,156.679
C01402=1064.513,382.170,389.589,174.823,35.711,156.680
C01403=1064.520,382.417,389.548,174.828,35.718,156.682
C01404=1064.527,382.664,389.509,174.833,35.725,156.683
C01405=1064.534,382.910,389.469,174.838,35.732,156.685
C01406=1064.541,383.157,389.428,174.843,35.738,156.687
C01407=1064.548,383.403,389.389,174.848,35.746,156.688
C01408=1064.556,383.649,389.349,174.853,35.753,156.690
C01409=1064.563,383.896,389.308,174.858,35.759,156.692
C01410=1064.571,384.143,389.268,174.863,35.767,156.693
C01411=1064.578,384.389,389.229,174.869,35.774,156.695
C01412=1064.585,384.637,389.188,174.873,35.781,156.697
C01413=1064.592,384.883,389.149,174.878,35.788,156.698
C01414=1064.599,385.129,389.107,174.883,35.795,156.700
C01415=1064.606,385.376,389.068,174.889,35.802,156.702
C01416=1064.614,385.623,389.028,174.894,35.809,156.703
C01417=1064.621,385.869,388.987,174.898,35.816,156.705
C01418=1064.628,386.115,388.947,174.904,35.823,156.707
C01419=1064.637,386.394,388.901,174.910,35.831,156.708
C01420=1064.644,386.672,388.856,174.915,35.839,156.710
C01421=1064.653,386.949,388.811,174.921,35.848,156.712
C01422=1064.661,387.227,388.765,174.927,35.856,156.714
C01423=1064.669,387.474,388.725,174.932,35.863,156.716
C01424=1064.676,387.720,388.684,174.938,35.870,156.718
C01425=1064.684,387.966,388.643,174.943,35.877,156.719
C01426=1064.691,388.213,388.603,174.948,35.885,156.721
C01427=1064.699,388.460,388.562,174.953,35.892,156.723
C01428=1064.705,388.706,388.522,174.958,35.899,156.724
C01429=1064.713,388.952,388.481,174.964,35.906,156.726
C01430=1064.721,389.199,388.440,174.969,35.914,156.728
C01431=1064.728,389.446,388.400,174.974,35.921,156.730
C01432=1064.736,389.693,388.359,174.980,35.928,156.731
C01433=1064.743,389.938,388.319,174.985,35.936,156.733
C01434=1064.750,390.185,388.278,174.990,35.943,156.735
C01435=1064.758,390.432,388.238,174.995,35.951,156.737
C01436=1064.765,390.678,388.196,175.001,35.958,156.738
C01437=1064.773,390.925,388.156,175.006,35.966,156.740
C01438=1064.781,391.171,388.115,175.011,35.973,156.742
C01439=1064.787,391.417,388.074,175.017,35.981,156.744
C01440=1064.795,391.663,388.033,175.022,35.988,156.745
C01441=1064.803,391.910,387.992,175.028,35.996,156.747
C01442=1064.810,392.156,387.951,175.033,36.003,156.749
C01443=1064.817,392.403,387.909,175.039,36.011,156.751
C01444=1064.825,392.649,387.869,175.044,36.019,156.753
C01445=1064.833,392.895,387.827,175.050,36.026,156.755
C01446=1064.840,393.142,387.786,175.055,36.034,156.756
C01447=1064.847,393.389,387.744,175.061,36.042,156.758
C01448=1064.855,393.635,387.704,175.066,36.049,156.760
C01449=1064.863,393.881,387.662,175.072,36.057,156.762
C01450=1064.870,394.127,387.621,175.077,36.065,156.764
C01451=1064.878,394.374,387.579,175.083,36.072,156.766
C01452=1064.885,394.621,387.538,175.088,36.080,156.768
C01453=1064.893,394.867,387.496,175.094,36.088,156.769
C01454=1064.900,395.113,387.455,175.099,36.096,156.771
C01455=1064.907,395.360,387.414,175.105,36.104,156.773
C01456=1064.915,395.606,387.372,175.110,36.111,156.775
C01457=1064.922,395.852,387.330,175.116,36.120,156.777
C01458=1064.930,396.098,387.289,175.121,36.127,156.779
C01459=1064.938,396.345,387.248,175.127,36.135,156.781
C01460=1064.945,396.590,387.206,175.132,36.143,156.783
C01461=1064.953,396.838,387.164,175.138,36.151,156.785
C01462=1064.961,397.084,387.122,175.144,36.159,156.786
C01463=1064.968,397.330,387.081,175.149,36.167,156.788
C01464=1064.976,397.576,387.039,175.155,36.175,156.790
C01465=1064.984,397.823,386.997,175.160,36.183,156.792
C01466=1064.991,398.070,386.956,175.166,36.191,156.794
C01467=1064.999,398.316,386.914,175.172,36.199,156.796
C01468=1065.005,398.562,386.871,175.177,36.207,156.798
C01469=1065.013,398.808,386.829,175.183,36.215,156.800
C01470=1065.021,399.055,386.787,175.188,36.223,156.802
C01471=1065.029,399.301,386.746,175.194,36.232,156.804
C01472=1065.036,399.547,386.704,175.201,36.240,156.806
C01473=1065.044,399.793,386.662,175.206,36.248,156.808
C01474=1065.051,400.040,386.619,175.212,36.256,156.810
C01475=1065.060,400.334,386.569,175.219,36.266,156.812
C01476=1065.070,400.628,386.518,175.225,36.276,156.815
C01477=1065.079,400.922,386.468,175.233,36.286,156.817
C01478=1065.088,401.217,386.417,175.239,36.296,156.820
C01479=1065.096,401.463,386.375,175.245,36.304,156.822
C01480=1065.104,401.710,386.333,175.252,36.313,156.824
C01481=1065.111,401.955,386.290,175.258,36.321,156.826
C01482=1065.120,402.202,386.248,175.263,36.329,156.828
C01483=1065.127,402.448,386.206,175.269,36.338,156.830
C01484=1065.135,402.695,386.163,175.275,36.346,156.832
C01485=1065.143,402.940,386.120,175.281,36.355,156.834
C01486=1065.151,403.187,386.078,175.287,36.363,156.836
C01487=1065.158,403.433,386.036,175.293,36.372,156.838
C01488=1065.166,403.679,385.992,175.299,36.380,156.840
C01489=1065.174,403.925,385.950,175.305,36.389,156.842
C01490=1065.181,404.172,385.907,175.311,36.397,156.844
C01491=1065.189,404.418,385.865,175.317,36.406,156.847
C01492=1065.197,404.664,385.822,175.323,36.415,156.849
C01493=1065.204,404.910,385.779,175.329,36.423,156.851
C01494=1065.213,405.156,385.736,175.335,36.432,156.853
C01495=1065.220,405.403,385.693,175.342,36.441,156.855
C01496=1065.228,405.649,385.651,175.348,36.450,156.857
C01497=1065.236,405.896,385.608,175.353,36.458,156.859
C01498=1065.244,406.142,385.565,175.359,36.467,156.862
C01499=1065.251,406.387,385.521,175.366,36.476,156.864
C01500=1065.259,406.634,385.478,175.372,36.485,156.866
C01501=1065.267,406.880,385.435,175.378,36.494,156.868
C01502=1065.275,407.126,385.392,175.385,36.502,156.870
C01503=1065.282,407.372,385.349,175.391,36.511,156.873
C01504=1065.291,407.618,385.306,175.397,36.521,156.875
C01505=1065.299,407.865,385.262,175.404,36.529,156.877
C01506=1065.306,408.110,385.219,175.409,36.538,156.879
C01507=1065.314,408.356,385.176,175.415,36.547,156.882
C01508=1065.322,408.603,385.132,175.422,36.556,156.884
C01509=1065.330,408.849,385.088,175.428,36.566,156.886
C01510=1065.338,409.095,385.046,175.434,36.575,156.888
C01511=1065.345,409.341,385.002,175.441,36.584,156.891
C01512=1065.353,409.587,384.958,175.447,36.593,156.893
C01513=1065.362,409.833,384.915,175.454,36.602,156.895
C01514=1065.370,410.079,384.871,175.460,36.611,156.897
C01515=1065.377,410.325,384.827,175.466,36.620,156.900
C01516=1065.386,410.571,384.784,175.473,36.630,156.902
C01517=1065.394,410.817,384.740,175.480,36.639,156.904
C01518=1065.402,411.064,384.697,175.487,36.648,156.907
C01519=1065.410,411.310,384.653,175.493,36.658,156.909
C01520=1065.418,411.555,384.609,175.499,36.667,156.911
C01521=1065.426,411.802,384.566,175.506,36.676,156.914
C01522=1065.434,412.047,384.521,175.512,36.685,156.916
C01523=1065.442,412.294,384.478,175.519,36.695,156.918
C01524=1065.451,412.539,384.434,175.525,36.704,156.921
C01525=1065.459,412.786,384.390,175.532,36.714,156.923
C01526=1065.467,413.031,384.346,175.539,36.723,156.925
C01527=1065.475,413.277,384.302,175.546,36.733,156.928
C01528=1065.483,413.523,384.258,175.552,36.742,156.930
C01529=1065.491,413.769,384.214,175.559,36.751,156.933
C01530=1065.499,414.015,384.170,175.565,36.761,156.935
C01531=1065.509,414.315,384.117,175.574,36.773,156.938
C01532=1065.519,414.613,384.063,175.582,36.784,156.941
C01533=1065.530,414.912,384.008,175.590,36.796,156.944
C01534=1065.539,415.210,383.955,175.599,36.808,156.947
C01535=1065.547,415.456,383.910,175.605,36.818,156.949
C01536=1065.556,415.702,383.866,175.612,36.828,156.952
C01537=1065.564,415.948,383.821,175.619,36.837,156.954
C01538=1065.572,416.194,383.777,175.626,36.847,156.957
C01539=1065.580,416.440,383.732,175.633,36.857,156.960
C01540=1065.588,416.686,383.688,175.639,36.867,156.962
C01541=1065.596,416.932,383.643,175.647,36.877,156.965
C01542=1065.604,417.178,383.599,175.654,36.887,156.967
C01543=1065.613,417.423,383.553,175.660,36.897,156.970
C01544=1065.621,417.670,383.509,175.668,36.907,156.972
C01545=1065.630,417.915,383.464,175.675,36.917,156.975
C01546=1065.638,418.161,383.419,175.681,36.927,156.977
C01547=1065.646,418.407,383.374,175.689,36.937,156.980
C01548=1065.654,418.652,383.329,175.696,36.947,156.982
C01549=1065.662,418.898,383.285,175.704,36.957,156.985
C01550=1065.671,419.145,383.240,175.710,36.967,156.988
C01551=1065.679,419.390,383.195,175.718,36.978,156.990
C01552=1065.688,419.636,383.150,175.725,36.988,156.993
C01553=1065.696,419.881,383.105,175.731,36.999,156.996
C01554=1065.705,420.127,383.059,175.739,37.009,156.998
C01555=1065.713,420.373,383.015,175.746,37.019,157.001
C01556=1065.722,420.619,382.969,175.754,37.029,157.004
C01557=1065.731,420.865,382.924,175.761,37.040,157.006
C01558=1065.738,421.110,382.878,175.768,37.050,157.009
C01559=1065.747,421.356,382.833,175.775,37.061,157.012
C01560=1065.755,421.602,382.787,175.783,37.071,157.014
C01561=1065.764,421.848,382.743,175.791,37.082,157.017
C01562=1065.772,422.093,382.698,175.798,37.092,157.020
C01563=1065.780,422.339,382.652,175.806,37.103,157.023
C01564=1065.789,422.585,382.606,175.812,37.113,157.025
C01565=1065.797,422.830,382.560,175.820,37.124,157.028
C01566=1065.806,423.076,382.514,175.828,37.135,157.031
C01567=1065.814,423.322,382.468,175.835,37.146,157.034
C01568=1065.823,423.567,382.423,175.843,37.156,157.036
C01569=1065.831,423.813,382.377,175.850,37.167,157.039
C01570=1065.840,424.058,382.331,175.858,37.178,157.042
C01571=1065.848,424.304,382.285,175.866,37.189,157.045
C01572=1065.857,424.550,382.240,175.874,37.200,157.048
C01573=1065.865,424.795,382.193,175.881,37.210,157.051
C01574=1065.874,425.041,382.148,175.889,37.221,157.053
C01575=1065.883,425.286,382.101,175.897,37.232,157.056
C01576=1065.892,425.532,382.056,175.904,37.243,157.059
C01577=1065.900,425.778,382.009,175.912,37.254,157.062
C01578=1065.909,426.023,381.964,175.920,37.265,157.065
C01579=1065.917,426.268,381.917,175.928,37.277,157.068
C01580=1065.926,426.514,381.872,175.936,37.288,157.071
C01581=1065.935,426.760,381.825,175.943,37.299,157.074
C01582=1065.944,427.005,381.779,175.951,37.310,157.077
C01583=1065.952,427.251,381.733,175.959,37.321,157.080
C01584=1065.961,427.497,381.686,175.967,37.332,157.083
C01585=1065.970,427.742,381.640,175.975,37.344,157.086
C01586=1065.979,427.987,381.593,175.984,37.355,157.089
C01587=1065.990,428.306,381.533,175.993,37.370,157.093
C01588=1066.001,428.625,381.472,176.004,37.385,157.096
C01589=1066.013,428.943,381.411,176.015,37.400,157.100
C01590=1066.024,429.261,381.351,176.026,37.415,157.104
C01591=1066.033,429.507,381.304,176.033,37.426,157.107
C01592=1066.042,429.753,381.257,176.041,37.438,157.110
C01593=1066.051,429.998,381.211,176.049,37.450,157.114
C01594=1066.060,430.243,381.163,176.058,37.461,157.117
C01595=1066.069,430.489,381.117,176.067,37.473,157.120
C01596=1066.077,430.734,381.070,176.075,37.485,157.123
C01597=1066.087,430.980,381.022,176.083,37.496,157.126
C01598=1066.095,431.225,380.975,176.092,37.508,157.129
C01599=1066.104,431.470,380.928,176.100,37.520,157.132
C01600=1066.113,431.716,380.881,176.108,37.532,157.136
C01601=1066.122,431.961,380.833,176.117,37.544,157.139
C01602=1066.131,432.206,380.786,176.125,37.556,157.142
C01603=1066.139,432.452,380.739,176.134,37.568,157.145
C01604=1066.149,432.697,380.691,176.142,37.580,157.148
C01605=1066.158,432.942,380.644,176.151,37.592,157.152
C01606=1066.167,433.187,380.597,176.160,37.604,157.155
C01607=1066.176,433.433,380.549,176.168,37.616,157.158
C01608=1066.185,433.678,380.501,176.177,37.629,157.162
C01609=1066.194,433.922,380.454,176.185,37.641,157.165
C01610=1066.203,434.168,380.406,176.195,37.653,157.168
C01611=1066.212,434.413,380.359,176.203,37.665,157.171
C01612=1066.221,434.659,380.311,176.212,37.677,157.175
C01613=1066.230,434.903,380.263,176.220,37.690,157.178
C01614=1066.239,435.149,380.215,176.230,37.703,157.182
C01615=1066.248,435.394,380.167,176.238,37.715,157.185
C01616=1066.258,435.639,380.119,176.247,37.727,157.188
C01617=1066.267,435.885,380.071,176.257,37.740,157.192
C01618=1066.276,436.130,380.024,176.265,37.753,157.195
C01619=1066.286,436.375,379.975,176.275,37.765,157.199
C01620=1066.295,436.620,379.928,176.283,37.778,157.202
C01621=1066.304,436.865,379.879,176.293,37.790,157.205
C01622=1066.313,437.110,379.831,176.302,37.803,157.209
C01623=1066.323,437.355,379.782,176.310,37.816,157.212
C01624=1066.332,437.600,379.735,176.320,37.829,157.216
C01625=1066.341,437.845,379.686,176.329,37.842,157.219
C01626=1066.351,438.090,379.638,176.339,37.855,157.223
C01627=1066.360,438.336,379.589,176.347,37.867,157.227
C01628=1066.369,438.580,379.541,176.357,37.881,157.230
C01629=1066.379,438.825,379.493,176.367,37.893,157.234
C01630=1066.388,439.071,379.444,176.376,37.907,157.237
C01631=1066.398,439.316,379.395,176.386,37.919,157.241
C01632=1066.407,439.561,379.347,176.394,37.933,157.245
C01633=1066.416,439.806,379.297,176.404,37.946,157.248
C01634=1066.426,440.051,379.249,176.414,37.959,157.252
C01635=1066.434,440.295,379.200,176.423,37.973,157.255
C01636=1066.445,440.540,379.151,176.433,37.986,157.259
C01637=1066.454,440.785,379.102,176.443,37.999,157.263
C01638=1066.463,441.030,379.053,176.452,38.013,157.267
C01639=1066.473,441.274,379.004,176.462,38.026,157.270
C01640=1066.482,441.520,378.955,176.472,38.040,157.274
C01641=1066.492,441.764,378.905,176.482,38.053,157.278
C01642=1066.502,442.010,378.856,176.492,38.067,157.282
C01643=1066.511,442.252,378.807,176.501,38.080,157.285
C01644=1066.521,442.495,378.759,176.511,38.094,157.289
C01645=1066.530,442.737,378.710,176.521,38.108,157.293
C01646=1066.540,442.979,378.661,176.531,38.121,157.297
C01647=1066.550,443.222,378.612,176.541,38.135,157.301
C01648=1066.559,443.465,378.562,176.551,38.149,157.305
C01649=1066.569,443.707,378.513,176.561,38.162,157.308
C01650=1066.579,443.949,378.464,176.571,38.176,157.312
C01651=1066.588,444.194,378.414,176.581,38.190,157.316
C01652=1066.597,444.439,378.364,176.591,38.204,157.320
C01653=1066.608,444.684,378.315,176.602,38.219,157.324
C01654=1066.617,444.929,378.265,176.612,38.233,157.328
C01655=1066.627,445.173,378.215,176.622,38.247,157.332
C01656=1066.637,445.418,378.166,176.632,38.261,157.336
C01657=1066.647,445.662,378.115,176.643,38.276,157.340
C01658=1066.657,445.908,378.065,176.653,38.290,157.344
C01659=1066.666,446.152,378.015,176.665,38.304,157.348
C01660=1066.677,446.397,377.965,176.675,38.318,157.352
C01661=1066.686,446.641,377.915,176.685,38.333,157.357
C01662=1066.697,446.886,377.864,176.696,38.348,157.361
C01663=1066.706,447.131,377.814,176.706,38.362,157.365
C01664=1066.716,447.375,377.764,176.718,38.377,157.369
C01665=1066.727,447.619,377.713,176.728,38.391,157.373
C01666=1066.736,447.863,377.663,176.739,38.406,157.377
C01667=1066.747,448.107,377.613,176.750,38.420,157.382
C01668=1066.760,448.350,377.564,176.761,38.434,157.386
C01669=1066.772,448.595,377.516,176.772,38.448,157.390
C01670=1066.787,448.840,377.468,176.783,38.462,157.393
C01671=1066.801,449.085,377.421,176.794,38.475,157.397
C01672=1066.817,449.330,377.374,176.804,38.488,157.401
C01673=1066.834,449.575,377.328,176.814,38.500,157.404
C01674=1066.853,449.820,377.284,176.824,38.512,157.408
C01675=1066.511,449.824,377.021,176.813,38.641,157.443
C01676=1066.492,449.579,377.066,176.803,38.629,157.439
C01677=1066.475,449.334,377.112,176.793,38.617,157.436
C01678=1066.459,449.089,377.159,176.783,38.604,157.432
C01679=1066.443,448.844,377.206,176.772,38.592,157.428
C01680=1066.430,448.599,377.253,176.761,38.578,157.424
C01681=1066.416,448.355,377.302,176.750,38.564,157.420
C01682=1066.404,448.110,377.351,176.739,38.550,157.416
C01683=1066.393,447.868,377.400,176.728,38.536,157.412
C01684=1066.383,447.623,377.451,176.716,38.521,157.408
C01685=1066.374,447.379,377.501,176.706,38.507,157.404
C01686=1066.363,447.134,377.552,176.695,38.492,157.400
C01687=1066.353,446.890,377.602,176.685,38.477,157.395
C01688=1066.343,446.645,377.653,176.673,38.463,157.391
C01689=1066.333,446.401,377.702,176.663,38.449,157.387
C01690=1066.323,446.156,377.753,176.652,38.434,157.383
C01691=1066.313,445.912,377.803,176.642,38.420,157.379
C01692=1066.303,445.667,377.854,176.631,38.405,157.375
C01693=1066.293,445.423,377.903,176.621,38.391,157.371
C01694=1066.283,445.177,377.953,176.610,38.377,157.367
C01695=1066.274,444.933,378.003,176.599,38.363,157.363
C01696=1066.263,444.689,378.053,176.589,38.349,157.359
C01697=1066.253,444.443,378.103,176.578,38.335,157.355
C01698=1066.244,444.199,378.153,176.568,38.321,157.351
C01699=1066.235,443.954,378.203,176.558,38.307,157.347
C01700=1066.225,443.726,378.249,176.549,38.294,157.343
C01701=1066.216,443.499,378.295,176.539,38.281,157.340
C01702=1066.207,443.272,378.341,176.530,38.268,157.336
C01703=1066.198,443.044,378.388,176.521,38.255,157.332
C01704=1066.189,442.816,378.434,176.511,38.242,157.329
C01705=1066.180,442.589,378.480,176.502,38.230,157.325
C01706=1066.171,442.361,378.526,176.492,38.217,157.322
C01707=1066.160,442.090,378.580,176.481,38.202,157.317
C01708=1066.150,441.845,378.629,176.471,38.188,157.314
C01709=1066.141,441.600,378.679,176.461,38.175,157.310
C01710=1066.131,441.356,378.728,176.451,38.161,157.306
C01711=1066.122,441.111,378.777,176.442,38.148,157.302
C01712=1066.112,440.866,378.826,176.432,38.134,157.298
C01713=1066.103,440.621,378.875,176.422,38.121,157.295
C01714=1066.093,440.376,378.924,176.412,38.108,157.291
C01715=1066.084,440.131,378.973,176.403,38.095,157.287
C01716=1066.074,439.886,379.022,176.393,38.081,157.284
C01717=1066.064,439.641,379.071,176.383,38.068,157.280
C01718=1066.055,439.396,379.120,176.374,38.055,157.276
C01719=1066.046,439.151,379.169,176.364,38.042,157.273
C01720=1066.037,438.906,379.217,176.354,38.029,157.269
C01721=1066.027,438.662,379.266,176.345,38.015,157.266
C01722=1066.018,438.417,379.314,176.335,38.003,157.262
C01723=1066.009,438.171,379.363,176.327,37.989,157.258
C01724=1065.999,437.926,379.411,176.317,37.977,157.255
C01725=1065.989,437.681,379.460,176.308,37.964,157.251
C01726=1065.980,437.436,379.508,176.298,37.951,157.248
C01727=1065.971,437.191,379.556,176.289,37.938,157.244
C01728=1065.962,436.946,379.605,176.280,37.926,157.241
C01729=1065.952,436.701,379.653,176.271,37.913,157.237
C01730=1065.942,436.455,379.701,176.261,37.900,157.234
C01731=1065.933,436.211,379.749,176.253,37.888,157.230
C01732=1065.924,435.965,379.797,176.243,37.875,157.227
C01733=1065.914,435.720,379.845,176.234,37.863,157.224
C01734=1065.905,435.475,379.893,176.226,37.851,157.220
C01735=1065.896,435.230,379.941,176.216,37.838,157.217
C01736=1065.888,434.984,379.989,176.207,37.825,157.213
C01737=1065.878,434.739,380.037,176.199,37.813,157.210
C01738=1065.869,434.495,380.085,176.189,37.801,157.207
C01739=1065.860,434.249,380.133,176.181,37.788,157.203
C01740=1065.851,434.004,380.180,176.172,37.776,157.200
C01741=1065.841,433.759,380.228,176.163,37.764,157.197
C01742=1065.832,433.514,380.275,176.154,37.752,157.193
C01743=1065.823,433.268,380.323,176.145,37.740,157.190
C01744=1065.814,433.023,380.371,176.137,37.728,157.187
C01745=1065.805,432.778,380.418,176.128,37.716,157.184
C01746=1065.796,432.533,380.466,176.120,37.703,157.180
C01747=1065.787,432.287,380.513,176.111,37.691,157.177
C01748=1065.778,432.042,380.560,176.102,37.680,157.174
C01749=1065.769,431.797,380.608,176.094,37.668,157.171
C01750=1065.760,431.551,380.655,176.085,37.656,157.167
C01751=1065.752,431.306,380.702,176.077,37.644,157.164
C01752=1065.743,431.061,380.750,176.068,37.632,157.161
C01753=1065.734,430.815,380.797,176.060,37.620,157.158
C01754=1065.725,430.570,380.843,176.052,37.609,157.155
C01755=1065.716,430.325,380.891,176.043,37.597,157.152
C01756=1065.707,430.079,380.938,176.035,37.585,157.149
C01757=1065.697,429.834,380.985,176.027,37.573,157.145
C01758=1065.689,429.588,381.032,176.019,37.562,157.142
C01759=1065.680,429.343,381.078,176.010,37.551,157.139
C01760=1065.669,429.023,381.139,175.999,37.536,157.135
C01761=1065.657,428.702,381.200,175.988,37.521,157.131
C01762=1065.646,428.382,381.262,175.977,37.505,157.127
C01763=1065.635,428.062,381.323,175.968,37.491,157.123
C01764=1065.625,427.817,381.369,175.959,37.479,157.120
C01765=1065.617,427.571,381.416,175.951,37.468,157.117
C01766=1065.608,427.325,381.462,175.943,37.457,157.114
C01767=1065.600,427.079,381.508,175.935,37.446,157.111
C01768=1065.591,426.834,381.554,175.927,37.435,157.108
C01769=1065.582,426.589,381.601,175.919,37.423,157.105
C01770=1065.573,426.343,381.647,175.912,37.412,157.103
C01771=1065.565,426.097,381.693,175.903,37.401,157.100
C01772=1065.555,425.852,381.739,175.895,37.390,157.097
C01773=1065.547,425.606,381.785,175.887,37.379,157.094
C01774=1065.538,425.361,381.832,175.879,37.368,157.091
C01775=1065.529,425.115,381.878,175.872,37.357,157.088
C01776=1065.520,424.869,381.924,175.864,37.346,157.085
C01777=1065.512,424.623,381.970,175.856,37.336,157.082
C01778=1065.503,424.379,382.015,175.849,37.324,157.079
C01779=1065.495,424.133,382.062,175.841,37.314,157.077
C01780=1065.486,423.887,382.108,175.833,37.303,157.074
C01781=1065.478,423.641,382.154,175.825,37.292,157.071
C01782=1065.469,423.395,382.199,175.818,37.282,157.068
C01783=1065.461,423.150,382.245,175.810,37.271,157.065
C01784=1065.452,422.905,382.291,175.803,37.260,157.063
C01785=1065.443,422.659,382.337,175.795,37.250,157.060
C01786=1065.435,422.414,382.382,175.787,37.239,157.057
C01787=1065.427,422.167,382.428,175.780,37.228,157.054
C01788=1065.418,421.922,382.473,175.772,37.218,157.052
C01789=1065.409,421.676,382.518,175.766,37.207,157.049
C01790=1065.401,421.430,382.564,175.758,37.197,157.046
C01791=1065.393,421.185,382.609,175.750,37.186,157.043
C01792=1065.385,420.939,382.655,175.743,37.176,157.041
C01793=1065.376,420.694,382.701,175.735,37.166,157.038
C01794=1065.368,420.448,382.745,175.728,37.155,157.035
C01795=1065.359,420.202,382.791,175.720,37.145,157.033
C01796=1065.351,419.956,382.836,175.714,37.135,157.030
C01797=1065.342,419.710,382.881,175.706,37.124,157.027
C01798=1065.334,419.465,382.926,175.699,37.114,157.025
C01799=1065.325,419.219,382.971,175.692,37.104,157.022
C01800=1065.317,418.973,383.016,175.684,37.093,157.019
C01801=1065.308,418.727,383.061,175.678,37.083,157.017
C01802=1065.301,418.481,383.106,175.670,37.073,157.014
C01803=1065.292,418.235,383.152,175.663,37.063,157.012
C01804=1065.283,417.990,383.196,175.655,37.053,157.009
C01805=1065.275,417.744,383.240,175.649,37.043,157.006
C01806=1065.266,417.498,383.286,175.642,37.033,157.004
C01807=1065.258,417.252,383.330,175.634,37.023,157.001
C01808=1065.250,417.006,383.375,175.628,37.013,156.999
C01809=1065.241,416.761,383.420,175.621,37.004,156.996
C01810=1065.234,416.515,383.465,175.613,36.994,156.994
C01811=1065.226,416.269,383.509,175.607,36.983,156.991
C01812=1065.217,416.023,383.554,175.600,36.974,156.989
C01813=1065.209,415.777,383.598,175.592,36.964,156.986
C01814=1065.201,415.531,383.642,175.586,36.954,156.984
